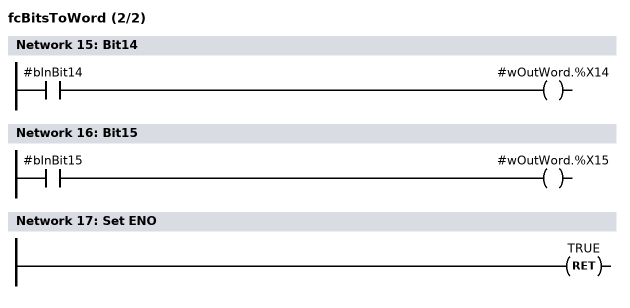
   RUNG wire#powerrail
      Contact( #bInBit14 )
      Coil( #wOutWord.%X14 )
   END_RUNG
   // the same network as SCL:
   #wOutWord.%X14 := #bInBit14;
END_REGION

REGION Network 16: Bit15
   RUNG wire#powerrail
      Contact( #bInBit15 )
      Coil( #wOutWord.%X15 )
   END_RUNG
   // the same network as SCL:
   #wOutWord.%X15 := #bInBit15;
END_REGION

REGION Network 17: Set ENO
   RUNG wire#powerrail
      ReturnCoil( TRUE )
   END_RUNG
   // the same network as SCL:
   ENO := TRUE;
   RETURN;
END_REGION
END_FUNCTION

FUNCTION_BLOCK "fbRoomFertigation"
{ S7_Optimized_Access := 'TRUE' }
VERSION : 0.1
   VAR_INPUT 
      arrInMutexRequests { ExternalAccessible := 'False'; ExternalVisible := 'False'; ExternalWritable := 'False'} : Array[0.."MAX_RACKS_PER_ROOM"] of Int;   // Array of mutex requests from racks
      arrInFertigationSettings { ExternalAccessible := 'False'; ExternalVisible := 'False'; ExternalWritable := 'False'} : Array[0.."MAX_RACKS_PER_ROOM"] of "udtFertigationSettings";
      rInTankLevel { ExternalAccessible := 'False'; ExternalVisible := 'False'; ExternalWritable := 'False'} : Real;
      rInNutrientALevel { ExternalAccessible := 'False'; ExternalVisible := 'False'; ExternalWritable := 'False'} : Real;
      rInNutrientBLevel { ExternalAccessible := 'False'; ExternalVisible := 'False'; ExternalWritable := 'False'} : Real;
      rInNutrientAcidLevel { ExternalAccessible := 'False'; ExternalVisible := 'False'; ExternalWritable := 'False'} : Real;
      rInpHSensor { ExternalAccessible := 'False'; ExternalVisible := 'False'; ExternalWritable := 'False'} : Real;
      rInECSensor { ExternalAccessible := 'False'; ExternalVisible := 'False'; ExternalWritable := 'False'} : Real;
      rInISESensor { ExternalAccessible := 'False'; ExternalVisible := 'False'; ExternalWritable := 'False'} : Real;
      rInORPReading { ExternalAccessible := 'False'; ExternalVisible := 'False'; ExternalWritable := 'False'} : Real;
      iInNumRacks { ExternalAccessible := 'False'; ExternalVisible := 'False'; ExternalWritable := 'False'} : Int;   // Number of racks to process mutex requests for
   END_VAR

   VAR_OUTPUT 
      bOutTankReturnSolenoid { ExternalAccessible := 'False'; ExternalVisible := 'False'; ExternalWritable := 'False'} : Bool;
      bOutMPathSolenoid { ExternalAccessible := 'False'; ExternalVisible := 'False'; ExternalWritable := 'False'} : Bool;
      bOutFreshWaterSolenoid { ExternalAccessible := 'False'; ExternalVisible := 'False'; ExternalWritable := 'False'} : Bool;
      bOutDischargeSolenoid { ExternalAccessible := 'False'; ExternalVisible := 'False'; ExternalWritable := 'False'} : Bool;
      bOutNutrientMixing { ExternalAccessible := 'False'; ExternalVisible := 'False'; ExternalWritable := 'False'} : Bool;
      bOutNutrientA { ExternalAccessible := 'False'; ExternalVisible := 'False'; ExternalWritable := 'False'} : Bool;
      bOutNutrientB { ExternalAccessible := 'False'; ExternalVisible := 'False'; ExternalWritable := 'False'} : Bool;
      bOutNutrientAcid { ExternalAccessible := 'False'; ExternalVisible := 'False'; ExternalWritable := 'False'} : Bool;
   END_VAR
   VAR_OUTPUT RETAIN
      arrOutNutrientReading { ExternalAccessible := 'False'; ExternalVisible := 'False'; ExternalWritable := 'False'} : Array[0.."MAX_RACKS_PER_ROOM"] of "udtNutrientReading";   // Array of nutrient readings going to racks
      arrOutMutexLocks { ExternalAccessible := 'False'; ExternalVisible := 'False'; ExternalWritable := 'False'} : Array[0.."MAX_RACKS_PER_ROOM"] of Int;   // Array of mutex locks going to racks
   END_VAR
   VAR_OUTPUT 
      arrOutSupplySolenoids { ExternalAccessible := 'False'; ExternalVisible := 'False'; ExternalWritable := 'False'} : Array[0.."MAX_RACKS_PER_ROOM"] of Bool;   // Array of supply solenoids for each rack
      arrOutReturnSolenoids { ExternalAccessible := 'False'; ExternalVisible := 'False'; ExternalWritable := 'False'} : Array[0.."MAX_RACKS_PER_ROOM"] of Bool;   // Array of return solenoids for each rack
   END_VAR

   VAR RETAIN
      Controls { ExternalVisible := 'False'} : Struct
         bPauseFertigation { ExternalVisible := 'False'} : Bool;   // While true, prevents next rack from locking
         rFloorPumpSpeedSP { ExternalVisible := 'False'} : Real;   // Floor pump speed (RPM)
         iNutrientMixingMode { ExternalVisible := 'False'} : Int;   // Nutrient mixing mode (0: off, 1: on, 2: 10 minute, 3: Continuous)
         rFreshLevelForMeasurementLoop { ExternalVisible := 'False'} : Real;   // Amount of fresh water to fill in the tank during rotate to clean measurement loop
         rFillLevelToPreviousShelf { ExternalVisible := 'False'} : Real := 8.0;   // Amount of water to push back to previous tank during return
         rReturnPathVolume { ExternalVisible := 'False'} : Real := 19.0;   // Return path volume (L) to fill from active rack
         rTankEmptyLevel { ExternalVisible := 'False'} : Real := 150.0;   // Volume at which tank is considered empty (L)
         rTankMaxVolume { ExternalVisible := 'False'} : Real := 900.0;   // Maximum volume for tank (L)
         bNutrientAgitation { ExternalVisible := 'False'} : Bool;
         tNutrientAgitationInterval { ExternalVisible := 'False'} : Time := T#60M;   // Agitation Frequency
         tNutrientAgitationDuration { ExternalVisible := 'False'} : Time := T#10M;   // Agitation Pump on-time
         rNutrientTanksLowerLimit { ExternalVisible := 'False'} : Real := 20.0;   // Liters
      END_STRUCT;
      Status { ExternalVisible := 'False'; ExternalWritable := 'False'} : Struct
         iState { ExternalVisible := 'False'; ExternalWritable := 'False'} : Int;   // Current operation (0: off, 1: Fill, 2:Measurement/Dosing, 3:Discharge)
         iActiveRack { ExternalVisible := 'False'; ExternalWritable := 'False'} : Int;   // Rack that currently has a lock, 0 if idle
         iLastMDRack { ExternalVisible := 'False'; ExternalWritable := 'False'} : Int;   // Keep track of previous rack for rotate and flush, 0 if previous operation was not measurement and dosing
      END_STRUCT;
      bTankReturnSolenoidCommand { ExternalAccessible := 'False'; ExternalVisible := 'False'; ExternalWritable := 'False'} : Bool;   // Command for tank return solenoid
      bMPathSolenoidCommand { ExternalAccessible := 'False'; ExternalVisible := 'False'; ExternalWritable := 'False'} : Bool;   // Command for measurement path solenoid
      bFreshWaterSolenoidCommand { ExternalAccessible := 'False'; ExternalVisible := 'False'; ExternalWritable := 'False'} : Bool;   // Command for fresh water solenoid
      bDischargeSolenoidCommand { ExternalAccessible := 'False'; ExternalVisible := 'False'; ExternalWritable := 'False'} : Bool;   // Command for discharge solenoid
      bNutrientMixingCommand { ExternalAccessible := 'False'; ExternalVisible := 'False'; ExternalWritable := 'False'} : Bool;   // Command for nutrient mixing enable
      bNutrientACommand { ExternalAccessible := 'False'; ExternalVisible := 'False'; ExternalWritable := 'False'} : Bool;   // Command for dosing nutrient A
      bNutrientBCommand { ExternalAccessible := 'False'; ExternalVisible := 'False'; ExternalWritable := 'False'} : Bool;   // Command for dosing nutrient B
      bNutrientAcidCommand { ExternalAccessible := 'False'; ExternalVisible := 'False'; ExternalWritable := 'False'} : Bool;
      TON_Discharge {InstructionName := 'TON_TIME'; LibVersion := '1.0'; S7_SetPoint := 'False'} : TON_TIME;
      TON_24HourNutrientMix {InstructionName := 'TON_TIME'; LibVersion := '1.0'; ExternalAccessible := 'False'; ExternalVisible := 'False'; ExternalWritable := 'False'; S7_SetPoint := 'False'} : TON_TIME;
   END_VAR
   VAR 
      fbRoomMeasurementDosing { ExternalAccessible := 'False'; ExternalVisible := 'False'; ExternalWritable := 'False'; S7_SetPoint := 'False'} : "fbRoomMeasurementDosing";
   END_VAR
   VAR RETAIN
      bTransferring { ExternalAccessible := 'False'; ExternalVisible := 'False'; ExternalWritable := 'False'} : Bool;   // Memory bit for transfer to rack during fill process
      rTransferredVolume { ExternalAccessible := 'False'; ExternalVisible := 'False'; ExternalWritable := 'False'} : Real;
      rVolumeToTransfer { ExternalAccessible := 'False'; ExternalVisible := 'False'; ExternalWritable := 'False'} : Real;
      bEndDischarge { ExternalAccessible := 'False'; ExternalVisible := 'False'; ExternalWritable := 'False'} : Bool;
   END_VAR
   VAR 
      TON_PeriodicNutrientAgitation {InstructionName := 'TON_TIME'; LibVersion := '1.0'} : TON_TIME;
      TP_PeriodicNutrientAgitation {InstructionName := 'TP_TIME'; LibVersion := '1.0'} : TP_TIME;
   END_VAR

   VAR_TEMP 
      bFoundActive : Bool;
      i : Int;   // Iterable for mutex request 
      tCurrentDateTime : Date_And_Time;   // Current PLC Date and Time
      tCurrentTime : Time_Of_Day;   // Current PLC Time of Day
      retVal : Int;   // Garbage return value from RD_LOC_T
      bMDDone : Bool;
      rTargetFillVolume : Real;
   END_VAR

   VAR CONSTANT 
      eRoomMode_Off : Int := 0;   // Room Off State
      eRoomMode_Fill : Int := 1;   // Room Filling State
      eRoomMode_MeasurementDosing : Int := 2;   // Room Measurement and Dosing State
      eRoomMode_Discharge : Int := 3;   // Room Discharge State
      eNutrientMixingMode_Off : Int := 0;   // Forced off
      eNutrientMixingMode_On : Int := 1;   // Forced on
      eNutrientMixingMode_Periodic : Int := 2;   // Run according to Interval/Duration settings
      eNutrientMixingMode_FullDay : Int := 3;   // Run for 24 hours then switch to Ten Minute mode
      MIX_START_TIME : Time_Of_Day := TOD#12:00:00;   // Start of 10 minute mix at noon
      MIX_END_TIME : Time_Of_Day := TOD#12:10:00;   // End of 10 minute mix at noon
   END_VAR


BEGIN
	REGION 0: Off
	    // Close all solenoids
	    // Iterate through mutex requests to trigger state change
	    // Send lock when mutex request arrives
	    
	    IF #Status.iState = #eRoomMode_Off THEN
	        #bTankReturnSolenoidCommand := 0;
	        #bMPathSolenoidCommand := 0;
	        #bFreshWaterSolenoidCommand := 0;
	        
	        #bFoundActive := 0;
	        IF NOT #Controls.bPauseFertigation THEN // if not paused, check for next rack requesting lock
	            FOR #i := 1 TO #iInNumRacks DO
	                IF #arrInMutexRequests[#i] <> #eRoomMode_Off THEN
	                    
	                    // Mutex request active - update state and active rack, send lock
	                    #Status.iState := #arrInMutexRequests[#i];
	                    #Status.iActiveRack := #i;
	                    #arrOutMutexLocks[#i] := #Status.iState;
	                    #bFoundActive := 1;
	                    //Break out of for loop
	                    EXIT;
	                END_IF;
	            END_FOR;
	        END_IF;
	        IF NOT #bFoundActive THEN
	            #Status.iActiveRack := 0;
	        END_IF;
	    END_IF;
	    
	    
	END_REGION
	
	REGION 1: Fill
	    // Open fresh water solenoid, fill until max volume reached or rack volume reached, close fresh water solenoid
	    // Open rack supply solenoid, activate floor pump, wait for main tank content to return to rack
	    
	    // Need to keep track of how much has been sent to the rack, until total volume added matches OperatingVolume + TotalShelfVolume or
	    // resevoir reaches max volume
	    
	    IF #Status.iState = #eRoomMode_Fill THEN
	        
	        #Status.iLastMDRack := 0; // no rotate if last rack last rack was filled
	        
	        #rTargetFillVolume := #arrInFertigationSettings[#Status.iActiveRack].rOperatingVolume
	        + #arrInFertigationSettings[#Status.iActiveRack].rTotalShelfVolume;
	        
	        IF #rTransferredVolume >= #rTargetFillVolume OR
	            #arrInFertigationSettings[#Status.iActiveRack].rRackCurrentVolume > #arrInFertigationSettings[#Status.iActiveRack].rMaxReservoirVolume THEN
	            // Full volume or rack reservoir is too full, done with fill
	            #Status.iState := #eRoomMode_Off;
	            #arrOutMutexLocks[#Status.iActiveRack] := 0;
	            
	            #arrOutSupplySolenoids[#Status.iActiveRack] := 0;
	            #bFreshWaterSolenoidCommand := 0;
	            
	            #bTransferring := 0;
	            #rTransferredVolume := 0;
	            
	            
	        ELSIF #rInTankLevel < #Controls.rTankMaxVolume AND
	            #rInTankLevel - #Controls.rTankEmptyLevel + #rTransferredVolume < #rTargetFillVolume AND
	            NOT #bTransferring THEN
	            // Adding water to the main tank
	            #bFreshWaterSolenoidCommand := 1;
	            
	        ELSIF NOT #bTransferring THEN
	            // Start transfer from main tank to rack
	            #bTransferring := 1;
	            #bFreshWaterSolenoidCommand := 0;
	            #rVolumeToTransfer := #rInTankLevel - #Controls.rTankEmptyLevel;
	            
	        END_IF;
	        
	        IF #bTransferring AND #rInTankLevel <= #Controls.rTankEmptyLevel THEN
	            // Transfer is done, add volume to transferred total
	            #bTransferring := 0;
	            #rTransferredVolume += #rVolumeToTransfer;
	            #rVolumeToTransfer := 0;
	            #arrOutSupplySolenoids[#Status.iActiveRack] := 0;
	            
	        END_IF;
	        
	        // Transfer from main tank to rack until main tank is empty
	        #arrOutSupplySolenoids[#Status.iActiveRack] := #bTransferring;
	        
	    END_IF;
	    
	    
	END_REGION
	
	
	REGION 2: Measurement AND Dosing
	    // Call measurement and dosing subfunction for the room
	    // Only write to outputs when in the correct mode
	    
	    // Reset the last rack id to skip rotate if that rack is not accepting rotate
	    IF #Status.iState = #eRoomMode_MeasurementDosing AND #Status.iLastMDRack <> 0 THEN
	        IF NOT #arrInFertigationSettings[#Status.iLastMDRack].bEnableIncomingRotate THEN
	            #Status.iLastMDRack := 0;
	        END_IF;
	    END_IF;
	    
	     #fbRoomMeasurementDosing(bInStart := (#Status.iState = #eRoomMode_MeasurementDosing),
	                              iInActiveRack := #Status.iActiveRack,
	                              iInPreviousRack := #Status.iLastMDRack,
	                              rInTankLevel := #rInTankLevel,
	                              rInRackLevel := #arrInFertigationSettings[#Status.iActiveRack].rRackCurrentVolume,
	                              rInISEReading := #rInISESensor,
	                              rInECReading := #rInECSensor,
	                              rInpHReading := #rInpHSensor,
	                              rInORPReading := #rInORPReading,
	                              rInFillLevelToPreviousShelf := #Controls.rFillLevelToPreviousShelf,
	                              rInFreshLevelForMLoop := #Controls.rFreshLevelForMeasurementLoop,
	                              rInReturnPathVolume := #Controls.rReturnPathVolume,
	                              rInTankEmptyLevel := #Controls.rTankEmptyLevel,
	                              InFertigationSettings := #arrInFertigationSettings[#Status.iActiveRack],
	                              bOutTankReturnSolenoidCommand => #fbRoomMeasurementDosing.bOutTankReturnSolenoidCommand,
	                              bOutActiveRackReturnSolenoidCommand => #fbRoomMeasurementDosing.bOutActiveRackReturnSolenoidCommand,
	                              bOutActiveRackSupplySolenoidCommand => #fbRoomMeasurementDosing.bOutActiveRackSupplySolenoidCommand,
	                              bOutPreviousRackReturnSolenoidCommand => #fbRoomMeasurementDosing.bOutPreviousRackReturnSolenoidCommand,
	                              bOutPreviousRackSupplySolenoidCommand => #fbRoomMeasurementDosing.bOutPreviousRackSupplySolenoidCommand,
	                              bOutFreshWaterSolenoidCommand => #fbRoomMeasurementDosing.bOutFreshWaterSolenoidCommand,
	                              bOutDischargeSolenoidCommand => #fbRoomMeasurementDosing.bOutDischargeSolenoidCommand,
	                              bOutMPathSolenoidCommand => #fbRoomMeasurementDosing.bOutMPathSolenoidCommand,
	                              bOutNutrientACommand => #fbRoomMeasurementDosing.bOutNutrientACommand,
	                              bOutNutrientBCommand => #fbRoomMeasurementDosing.bOutNutrientBCommand,
	                              OutNutrientReadings => #fbRoomMeasurementDosing.OutNutrientReadings,
	                              bOutDone => #bMDDone);
	    
	    //Handle output writing
	    IF #Status.iState = #eRoomMode_MeasurementDosing THEN
	        #bTankReturnSolenoidCommand := #fbRoomMeasurementDosing.bOutTankReturnSolenoidCommand;
	        #bFreshWaterSolenoidCommand := #fbRoomMeasurementDosing.bOutFreshWaterSolenoidCommand;
	        #bDischargeSolenoidCommand := #fbRoomMeasurementDosing.bOutDischargeSolenoidCommand;
	        #bMPathSolenoidCommand := #fbRoomMeasurementDosing.bOutMPathSolenoidCommand;
	        #bNutrientACommand := #fbRoomMeasurementDosing.bOutNutrientACommand;
	        #bNutrientBCommand := #fbRoomMeasurementDosing.bOutNutrientBCommand;
	        #arrOutReturnSolenoids[#Status.iActiveRack] := #fbRoomMeasurementDosing.bOutActiveRackReturnSolenoidCommand;
	        #arrOutSupplySolenoids[#Status.iActiveRack] := #fbRoomMeasurementDosing.bOutActiveRackSupplySolenoidCommand;
	        #arrOutReturnSolenoids[#Status.iLastMDRack] := #fbRoomMeasurementDosing.bOutPreviousRackReturnSolenoidCommand;
	        #arrOutSupplySolenoids[#Status.iLastMDRack] := #fbRoomMeasurementDosing.bOutPreviousRackSupplySolenoidCommand;
	        #arrOutNutrientReading[#Status.iActiveRack] := #fbRoomMeasurementDosing.OutNutrientReadings;
	        
	        IF #bMDDone THEN
	            #Status.iState := #eRoomMode_Off;
	            #arrOutMutexLocks[#Status.iActiveRack] := #eRoomMode_Off;
	            #Status.iLastMDRack := #Status.iActiveRack; // save rack id for rotate on next M&D
	        END_IF;
	    END_IF;
	    
	END_REGION
	
	REGION 3: Discharge
	    // Open discharge solenoid and rack's return solenoid
	    // Wait for discharge time
	    // Close solenoids and release lock
	    // Return to Off mode
	    
	    #TON_Discharge(IN := (#Status.iState = #eRoomMode_Discharge),
	                   PT := #arrInFertigationSettings[#Status.iActiveRack].tDischargeTime);
	    
	    IF #Status.iState = #eRoomMode_Discharge THEN
	        
	        IF #TON_Discharge.Q OR #arrInFertigationSettings[#Status.iActiveRack].bEndDischargeCommand THEN
	            #bEndDischarge := 1;
	        END_IF;
	        
	        
	        IF #bEndDischarge THEN
	            #arrOutMutexLocks[#Status.iActiveRack] := #eRoomMode_Off;
	            
	            // wait until pump stops to close valves
	            IF #arrInFertigationSettings[#Status.iActiveRack].bPumpAtStandstill THEN 
	                #bDischargeSolenoidCommand := 0;
	                #arrOutReturnSolenoids[#Status.iActiveRack] := 0;
	                #Status.iLastMDRack := 0; // no rotate if last rack was discharged
	                #Status.iState := #eRoomMode_Off;
	                #bEndDischarge := 0;
	                #TON_Discharge.IN := 0; // reset timer
	            END_IF;
	            
	        ELSE
	            #bDischargeSolenoidCommand := 1;
	            #arrOutReturnSolenoids[#Status.iActiveRack] := 1;
	            
	        END_IF;
	        
	    END_IF;
	    
	END_REGION
	
	REGION Nutrient Tank Mixing
	    // 0: forced off, 1: forced on, 2: 10 minutes per day at noon, 3: Run for 24 hours then jump to mode 2
	    
	    
	    // if the tanks are too low, switch agitation to off
	    (*IF #rInNutrientALevel < #Controls.rNutrientTanksLowerLimit OR #rInNutrientBLevel < #Controls.rNutrientTanksLowerLimit THEN
	        #Controls.iNutrientMixingMode := #eNutrientMixingMode_Off;
	    END_IF;
	    *)
	    
	    #TON_24HourNutrientMix(IN := (#Controls.iNutrientMixingMode = #eNutrientMixingMode_FullDay),
	                           PT := T#24h);
	    
	    // if mode is set to periodic agitation, run timer to periodically run pumps
	    #Controls.bNutrientAgitation := #TON_PeriodicNutrientAgitation.Q;
	    #TON_PeriodicNutrientAgitation(IN := #Controls.iNutrientMixingMode = #eNutrientMixingMode_Periodic AND NOT #Controls.bNutrientAgitation,
	                                   PT := #Controls.tNutrientAgitationInterval);
	    
	    #TP_PeriodicNutrientAgitation(IN := #Controls.bNutrientAgitation,
	                                  PT := #Controls.tNutrientAgitationDuration,
	                                  Q => #bNutrientMixingCommand);
	    
	    
	    IF #Controls.iNutrientMixingMode = #eNutrientMixingMode_Off THEN
	        #bNutrientMixingCommand := 0;
	        
	    ELSIF #Controls.iNutrientMixingMode = #eNutrientMixingMode_On THEN
	        #bNutrientMixingCommand := 1;
	        
	        (*
	    ELSIF #Controls.iNutrientMixingMode = #eNutrientMixingMode_Periodic THEN
	      
	        // Extract current PLC time
	        #retVal := RD_LOC_T(OUT => #tCurrentDateTime);
	        #tCurrentTime := DT_TO_TOD(IN := #tCurrentDateTime);
	        
	        IF (#tCurrentTime < #MIX_END_TIME) AND (#tCurrentTime > #MIX_START_TIME) T
	            #bNutrientMixingCommand := 1;
	        ELSE
	            #bNutrientMixingCommand := 0;
	        END_IF;
	        
	        *)
	        
	    ELSIF #Controls.iNutrientMixingMode = #eNutrientMixingMode_FullDay THEN
	        
	        IF #TON_24HourNutrientMix.Q THEN
	            #bNutrientMixingCommand := 0;
	            #Controls.iNutrientMixingMode := #eNutrientMixingMode_Periodic;
	        ELSE
	            #bNutrientMixingCommand := 1;
	        END_IF;
	        
	        // Catchall for incorrectly entered state, just turn off mixer
	    //ELSE
	    //    #bNutrientMixingCommand := 0;
	    END_IF;
	    
	    // IF not forced on and then tank levels are too low, override above and disable mixing until tanks are filled
	    IF NOT (#Controls.iNutrientMixingMode = #eNutrientMixingMode_On) AND
	           (#rInNutrientALevel < #Controls.rNutrientTanksLowerLimit OR
	            #rInNutrientBLevel < #Controls.rNutrientTanksLowerLimit) THEN
	        #bNutrientMixingCommand := 0;
	    END_IF;
	    
	END_REGION
	
	REGION Set digital outputs
	    #bOutTankReturnSolenoid := #bTankReturnSolenoidCommand;
	    #bOutMPathSolenoid      := #bMPathSolenoidCommand;
	    #bOutFreshWaterSolenoid := #bFreshWaterSolenoidCommand;
	    #bOutDischargeSolenoid  := #bDischargeSolenoidCommand;
	    #bOutNutrientMixing     := #bNutrientMixingCommand;
	    #bOutNutrientA          := #bNutrientACommand;
	    #bOutNutrientB          := #bNutrientBCommand;
	    #bOutNutrientAcid       := #bNutrientAcidCommand;
	    
	END_REGION
	
	
	
END_FUNCTION_BLOCK

FUNCTION_BLOCK "fbRoomMeasurementDosing"
{ S7_Optimized_Access := 'TRUE' }
VERSION : 0.1
   VAR_INPUT 
      bInStart { ExternalAccessible := 'False'; ExternalVisible := 'False'; ExternalWritable := 'False'} : Bool;   // Start command for sequence
      iInActiveRack { ExternalAccessible := 'False'; ExternalVisible := 'False'; ExternalWritable := 'False'} : Int;   // Current rack requesting MD
      iInPreviousRack { ExternalAccessible := 'False'; ExternalVisible := 'False'; ExternalWritable := 'False'} : Int;   // Previous rack, if last operation was also MD (0 otherwise)
      rInTankLevel { ExternalAccessible := 'False'; ExternalVisible := 'False'; ExternalWritable := 'False'} : Real;   // Current tank level (L)
      rInISEReading { ExternalAccessible := 'False'; ExternalVisible := 'False'; ExternalWritable := 'False'} : Real;   // Current ISE sensor level
      rInECReading { ExternalAccessible := 'False'; ExternalVisible := 'False'; ExternalWritable := 'False'} : Real;   // Current EC sensor level
      rInpHReading { ExternalAccessible := 'False'; ExternalVisible := 'False'; ExternalWritable := 'False'} : Real;   // Current pH sensor level
      rInORPReading { ExternalAccessible := 'False'; ExternalVisible := 'False'; ExternalWritable := 'False'} : Real;
      rInRackLevel { ExternalAccessible := 'False'; ExternalVisible := 'False'; ExternalWritable := 'False'} : Real;   // Current rack reservoir level
      rInFreshLevelForMLoop { ExternalAccessible := 'False'; ExternalVisible := 'False'; ExternalWritable := 'False'} : Real;
      rInFillLevelToPreviousShelf { ExternalAccessible := 'False'; ExternalVisible := 'False'; ExternalWritable := 'False'} : Real;
      rInReturnPathVolume { ExternalAccessible := 'False'; ExternalVisible := 'False'; ExternalWritable := 'False'} : Real;   // Return path volume (L) to fill from active rack
      rInTankEmptyLevel { ExternalAccessible := 'False'; ExternalVisible := 'False'; ExternalWritable := 'False'} : Real;   // Volume at which tank is considered empty (L)
      InFertigationSettings { ExternalAccessible := 'False'; ExternalVisible := 'False'; ExternalWritable := 'False'} : "udtFertigationSettings";   // Current rack fertigation settings
   END_VAR

   VAR_OUTPUT RETAIN
      bOutTankReturnSolenoidCommand { ExternalAccessible := 'False'; ExternalVisible := 'False'; ExternalWritable := 'False'} : Bool;   // Output for writing to tank return solenoid
      bOutActiveRackReturnSolenoidCommand { ExternalAccessible := 'False'; ExternalVisible := 'False'; ExternalWritable := 'False'} : Bool;
      bOutActiveRackSupplySolenoidCommand { ExternalAccessible := 'False'; ExternalVisible := 'False'; ExternalWritable := 'False'} : Bool;
      bOutPreviousRackReturnSolenoidCommand { ExternalAccessible := 'False'; ExternalVisible := 'False'; ExternalWritable := 'False'} : Bool;
      bOutPreviousRackSupplySolenoidCommand { ExternalAccessible := 'False'; ExternalVisible := 'False'; ExternalWritable := 'False'} : Bool;
      bOutFreshWaterSolenoidCommand { ExternalAccessible := 'False'; ExternalVisible := 'False'; ExternalWritable := 'False'} : Bool;
      bOutDischargeSolenoidCommand { ExternalAccessible := 'False'; ExternalVisible := 'False'; ExternalWritable := 'False'} : Bool;
      bOutMPathSolenoidCommand { ExternalAccessible := 'False'; ExternalVisible := 'False'; ExternalWritable := 'False'} : Bool;
      bOutNutrientACommand { ExternalAccessible := 'False'; ExternalVisible := 'False'; ExternalWritable := 'False'} : Bool;   // Output for writing to Nutrient A enable
      bOutNutrientBCommand { ExternalAccessible := 'False'; ExternalVisible := 'False'; ExternalWritable := 'False'} : Bool;   // Output for writing to Nutrient B enable
      OutNutrientReadings { ExternalAccessible := 'False'; ExternalVisible := 'False'; ExternalWritable := 'False'} : "udtNutrientReading";   // Final measured sensor levels for rack
      bOutDone { ExternalAccessible := 'False'; ExternalVisible := 'False'; ExternalWritable := 'False'} : Bool;
   END_VAR

   VAR RETAIN
      iState { ExternalAccessible := 'False'; ExternalVisible := 'False'; ExternalWritable := 'False'} : Int;
      iNextState { ExternalAccessible := 'False'; ExternalVisible := 'False'; ExternalWritable := 'False'} : Int;
      rTankStartingLevel { ExternalAccessible := 'False'; ExternalVisible := 'False'; ExternalWritable := 'False'} : Real;
      TON_MeasurementTimer {InstructionName := 'TON_TIME'; LibVersion := '1.0'; ExternalAccessible := 'False'; ExternalVisible := 'False'; ExternalWritable := 'False'; S7_SetPoint := 'False'} : TON_TIME;
      TON_NutrientATimer {InstructionName := 'TON_TIME'; LibVersion := '1.0'; ExternalAccessible := 'False'; ExternalVisible := 'False'; ExternalWritable := 'False'; S7_SetPoint := 'False'} : TON_TIME;
      TON_NutrientBTimer {InstructionName := 'TON_TIME'; LibVersion := '1.0'; ExternalAccessible := 'False'; ExternalVisible := 'False'; ExternalWritable := 'False'; S7_SetPoint := 'False'} : TON_TIME;
   END_VAR
   VAR 
      TON_TankLowLimitTimer {InstructionName := 'TON_TIME'; LibVersion := '1.0'} : TON_TIME;
   END_VAR

   VAR CONSTANT 
      eMDState_Idle : Int;
      eMDState_Rotate_Start : Int := 100;
      eMDState_Rotate_FillTankFromRack : Int := 102;
      eMDState_Rotate_PushToPrevious : Int := 104;
      eMDState_Rotate_FillTankFresh : Int := 106;
      eMDState_Rotate_MeasurementLoop : Int := 108;
      eMDState_Rotate_Done : Int := 119;
      eMDState_Measure_Start : Int := 120;
      eMDState_Measure_FillTankFromRack : Int := 122;
      eMDState_Measure_OpenMLoop : Int := 124;
      eMDState_Measure_Done : Int := 139;
      eMDState_Dosing_Start : Int := 140;
      eMDState_Dosing_AddNutrientA : Int := 142;
      eMDState_Dosing_AddNutrientB : Int := 144;
      eMDState_Dosing_AddFreshWater : Int := 146;
      eMDState_Dosing_Done : Int := 159;
      eMDState_Return_Start : Int := 160;
      eMDState_Return_FillPreviousRack : Int := 162;
      eMDState_Return_FillActiveRack : Int := 164;
      eMDState_Return_CloseSupplyPath : Int := 166;
      eMDState_Return_Done : Int := 169;
      iISEMode_Off : Int := 0;
      iISEMode_Load : Int := 1;
      iISEMode_Deplete : Int := 2;
   END_VAR


BEGIN
	REGION State 0: Idle
	    // Wait for start command to move on to rotate if a previous rack used the piping 
	    //  or directly to measure if not 
	    
	    IF #iState = #eMDState_Idle THEN
	        #bOutDone := 0;
	        IF #bInStart THEN
	            IF #iInPreviousRack = 0 OR #iInPreviousRack = #iInActiveRack THEN
	                #iNextState := #eMDState_Measure_Start;
	            ELSE
	                #iNextState := #eMDState_Rotate_Start;
	            END_IF;
	        END_IF;
	    END_IF;
	        
	    
	END_REGION
	
	REGION State 100: Rotate
	    // Open the tank return solenoid
	    // Open the return solenoid and close the shelf solenoid for the current rack until a fixed amount of water is pumped into the tank
	    // Close the return solenoid of the current rack and open the supply valve of the previous rack to push 19L from the 
	    //     tank into the previous rack. 
	    //     
	    
	    // Open tank return and rack return, close shelf, record starting tank level, then move to next state
	    IF #iState = #eMDState_Rotate_Start THEN
	        #bOutTankReturnSolenoidCommand := 1; 
	        #bOutActiveRackReturnSolenoidCommand := 1;
	        #iNextState := #eMDState_Rotate_FillTankFromRack;
	        #rTankStartingLevel := #rInTankLevel;
	    END_IF;
	    
	    // Once the target fill level is reached, close the return solenoids, open the previous rack's supply, then move to next state
	    IF #iState = #eMDState_Rotate_FillTankFromRack THEN
	        IF #rInTankLevel >= #rTankStartingLevel + #rInReturnPathVolume  OR #rInRackLevel <= #InFertigationSettings.rMinReservoirVolume THEN
	            #bOutActiveRackReturnSolenoidCommand := 0;
	            #bOutPreviousRackSupplySolenoidCommand := 1;
	            #bOutTankReturnSolenoidCommand := 1;
	            #iNextState := #eMDState_Rotate_PushToPrevious;
	        END_IF;
	    END_IF;
	    
	    // Run until 19L have been pushed into the previous rack and the tank is back at its original level, then close the
	    // previous rack's supply solenoid and move to next state
	    IF #iState = #eMDState_Rotate_PushToPrevious THEN
	        
	        IF #rInTankLevel <= #rTankStartingLevel * 1.2 THEN // HACK
	            #bOutPreviousRackSupplySolenoidCommand := 0;
	            #iNextState := #eMDState_Rotate_FillTankFresh;
	        END_IF;
	        
	    END_IF;
	    
	    // Open the fresh water supply and fill the tank until the target level is reached, then close the fresh water supply, open the
	    // measurement path solenoid and the discharge solenoid and move to the next state
	    IF #iState = #eMDState_Rotate_FillTankFresh THEN
	        
	        IF #rInTankLevel >= #rTankStartingLevel + #rInFreshLevelForMLoop THEN
	            #bOutFreshWaterSolenoidCommand := 0;
	            #bOutMPathSolenoidCommand := 1;
	            #bOutDischargeSolenoidCommand := 1;
	            #bOutTankReturnSolenoidCommand := 0;
	            #iNextState := #eMDState_Rotate_MeasurementLoop;
	        ELSE
	            #bOutFreshWaterSolenoidCommand := 1;
	        END_IF;
	    END_IF;
	    
	    // Push water out through the measurement loop. Once the tank is empty, close measurement path solenoid and
	    // the discharge solenoid and move to the next state
	    IF #iState = #eMDState_Rotate_MeasurementLoop THEN
	        
	        IF #rInTankLevel <= #rInTankEmptyLevel THEN
	            
	            #bOutMPathSolenoidCommand := 0;
	            #bOutDischargeSolenoidCommand := 0;
	            #iNextState := #eMDState_Rotate_Done;
	        END_IF;
	    END_IF;
	    
	    IF #iState = #eMDState_Rotate_Done THEN
	        #iNextState := #eMDState_Measure_Start;
	    END_IF;
	    
	END_REGION
	
	REGION State 120: Measure
	    // Receive water from rack and start measurement phase. Open measurement loop, push water through, record sensor readings, 
	    // determine setpoints, and move on to dosing
	    
	    #TON_MeasurementTimer(IN := (#iState = #eMDState_Measure_OpenMLoop),
	                         PT := #InFertigationSettings.tMeasurementTime);
	    
	    // Open tank return and shelf return solenoid
	    IF #iState = #eMDState_Measure_Start THEN
	        #bOutTankReturnSolenoidCommand := 1;
	        #bOutActiveRackReturnSolenoidCommand := 1;
	        #iNextState := #eMDState_Measure_FillTankFromRack;
	        #rTankStartingLevel := #rInTankLevel;
	    END_IF;
	    
	    // Wait to receive target level from rack, close rack return solenoid
	    IF #iState = #eMDState_Measure_FillTankFromRack THEN
	        IF #rInTankLevel >= (#InFertigationSettings.rMeasurementVolume + #rInTankEmptyLevel) OR
	            #rInRackLevel <= #InFertigationSettings.rMinReservoirVolume THEN
	            #iNextState := #eMDState_Measure_OpenMLoop;
	            #bOutActiveRackReturnSolenoidCommand := 0;
	        END_IF;
	    END_IF;
	    
	    // Open MPath solenoid, wait for measurement time then record measurement
	    IF #iState = #eMDState_Measure_OpenMLoop THEN
	        
	        IF #TON_MeasurementTimer.Q THEN
	            #OutNutrientReadings.rISEReading := #rInISEReading;
	            #OutNutrientReadings.rECReading := #rInECReading;
	            #OutNutrientReadings.rpHReading := #rInpHReading;
	            #OutNutrientReadings.rORPReading := #rInORPReading;
	            #bOutMPathSolenoidCommand := 0;
	            #bOutTankReturnSolenoidCommand := 0;
	            #iNextState := #eMDState_Measure_Done;
	        ELSE
	            #bOutMPathSolenoidCommand := 1;
	        END_IF;
	    END_IF;
	    
	    
	    IF #iState = #eMDState_Measure_Done THEN
	        #iNextState := #eMDState_Dosing_Start;
	    END_IF;
	   
	    
	END_REGION
	
	REGION State 140: Dosing
	    
	    // Check if rack fertigation logic has requested dosing
	    // Add enabled nutrients one at a time for dosing time then add fresh water to tank
	    
	    IF #iState = #eMDState_Dosing_Start THEN
	        
	        IF #InFertigationSettings.bDosingActive THEN
	            
	            IF #InFertigationSettings.bNutrientAEnable THEN
	                #iNextState := #eMDState_Dosing_AddNutrientA;
	            ELSIF #InFertigationSettings.bNutrientBEnable THEN
	                #iNextState := #eMDState_Dosing_AddNutrientB;
	            ELSE
	                #iNextState := #eMDState_Dosing_AddFreshWater;
	            END_IF;
	            
	        ELSE
	            #iNextState := #eMDState_Dosing_AddFreshWater;
	        END_IF;
	    END_IF;
	    
	    #TON_NutrientATimer(IN := (#iState = #eMDState_Dosing_AddNutrientA),
	                       PT := #InFertigationSettings.tNutrientDosingDuration);
	    // Add nutrient A for dosing time, then check if nutrient B is needed
	    IF #iState = #eMDState_Dosing_AddNutrientA THEN
	        
	        IF #TON_NutrientATimer.Q THEN
	            #bOutNutrientACommand := 0;
	            IF #InFertigationSettings.bNutrientBEnable THEN
	                #iNextState := #eMDState_Dosing_AddNutrientB;
	            ELSE
	                #iNextState := #eMDState_Dosing_AddFreshWater;
	            END_IF;
	        ELSE
	            #bOutNutrientACommand := 1;
	        END_IF;
	    END_IF;
	    
	    #TON_NutrientBTimer(IN := (#iState = #eMDState_Dosing_AddNutrientB),
	                       PT := #InFertigationSettings.tNutrientDosingDuration);
	    // Add nutrient B for dosing time, then move on to water fill
	    IF #iState = #eMDState_Dosing_AddNutrientB THEN
	        
	        IF #TON_NutrientBTimer.Q THEN
	            #bOutNutrientBCommand := 0;
	            #iNextState := #eMDState_Dosing_AddFreshWater;
	        ELSE
	            #bOutNutrientBCommand := 1;
	        END_IF;
	    END_IF;
	    
	    // Add fresh water to tank if tank level plus rack is less than the operating volume
	    IF #iState = #eMDState_Dosing_AddFreshWater THEN
	        IF (#rInTankLevel - #rInTankEmptyLevel + #rInRackLevel < #InFertigationSettings.rOperatingVolume) THEN
	            #bOutFreshWaterSolenoidCommand := 1;
	        ELSE
	            #bOutFreshWaterSolenoidCommand := 0;
	            #iNextState := #eMDState_Dosing_Done;
	        END_IF;
	    END_IF;
	    
	    
	    IF #iState = #eMDState_Dosing_Done THEN
	        #iNextState := #eMDState_Return_Start;
	    END_IF;
	    
	END_REGION
	
	REGION State 160: Return TO Tank
	    // If a previous rack was used, open supply path to previous rack, wait for 8L drop in tank
	    // Open supply path to active rack, activate floor pump, wait for tank contents to return to rack
	    // Close supply path
	    
	    // Determine which rack to start return to
	    IF #iState = #eMDState_Return_Start THEN
	        
	        IF #iInPreviousRack = 0 OR #iInPreviousRack = #iInActiveRack  THEN
	            #iNextState := #eMDState_Return_FillActiveRack;
	        ELSE
	            #iNextState := #eMDState_Return_FillPreviousRack;
	        END_IF;
	        #rTankStartingLevel := #rInTankLevel;
	    END_IF;
	    
	    // Open supply path to previous rack, wait for 8L drop in tank, close previous rack return path
	    IF #iState = #eMDState_Return_FillPreviousRack THEN
	        #bOutPreviousRackSupplySolenoidCommand := 1;
	        IF #rInTankLevel < (#rTankStartingLevel - #rInFillLevelToPreviousShelf) THEN
	            #bOutPreviousRackSupplySolenoidCommand := 0;
	            #iNextState := #eMDState_Return_FillActiveRack;
	        END_IF;
	    END_IF;
	    
	    // Open supply path to active rack
	    IF #iState = #eMDState_Return_FillActiveRack THEN
	        #rTankStartingLevel := #rInTankLevel;
	        #bOutActiveRackSupplySolenoidCommand := 1;
	        #iNextState := #eMDState_Return_CloseSupplyPath;
	    END_IF;
	    
	    // Wait for tank to empty, close supply path
	    //#TON_TankLowLimitTimer(IN:=#rInTankLevel <= #rInTankEmptyLevel,
	    //                       PT:=T#3s);
	    IF #iState = #eMDState_Return_CloseSupplyPath THEN
	        IF #rInTankLevel <= #rInTankEmptyLevel * 1.2 OR #rInRackLevel >= #InFertigationSettings.rMaxReservoirVolume THEN // HACK
	            #bOutActiveRackSupplySolenoidCommand := 0;
	            #iNextState := #eMDState_Return_Done;
	        END_IF;
	    END_IF;
	    
	    //Return to Idle at end of M&D
	    IF #iState = #eMDState_Return_Done THEN
	        #bOutDone := 1;
	        #iNextState := #eMDState_Idle;
	    END_IF;
	    
	END_REGION
	
	
	REGION Update State
	    IF #iState <> #iNextState THEN
	        #iState := #iNextState;
	    END_IF;
	END_REGION
	
	
END_FUNCTION_BLOCK

FUNCTION_BLOCK "fbRoomHVAC"   // FB2, LAD
{ S7_Optimized_Access := 'TRUE' }
VERSION : 0.1
// stored: AutoNumber true, IsIECCheckEnabled false, IsRetainMemResEnabled false, MemoryReserve 100, SetENOAutomatically false, UDAEnableTagReadback false
   VAR_INPUT
      iInCO2ReadingRaw { ExternalAccessible := 'False'; ExternalVisible := 'False'; ExternalWritable := 'False'} : Int;
   END_VAR
   VAR_OUTPUT
      bOutCO2Solenoid { ExternalAccessible := 'False'; ExternalVisible := 'False'; ExternalWritable := 'False'} : Bool;
   END_VAR
   VAR
      Temperature_Cooling { ExternalVisible := 'False'} : "fbAlarmedSetpoint";
      Humidity { ExternalVisible := 'False'} : "fbAlarmedSetpoint";
   END_VAR
   VAR RETAIN
      Controls { ExternalVisible := 'False'} : Struct
         rHeatingSP { ExternalVisible := 'False'} : Real := 55.0;
         bResetAlarm { ExternalVisible := 'False'} : Bool;
         bResetModbus { ExternalVisible := 'False'} : Bool;
         rDehum_SAT_SP { ExternalVisible := 'False'} : Real := 65.0;
         rDehum_MOD_SP { ExternalVisible := 'False'} : Real := 60.0;
      END_STRUCT;
      Status { ExternalVisible := 'False'; ExternalWritable := 'False'} : Struct
         SupplyAirTemperature { ExternalVisible := 'False'; ExternalWritable := 'False'} : Real;
         bModbusError { ExternalVisible := 'False'; ExternalWritable := 'False'} : Bool;
         wLastModbusErrorCode { ExternalVisible := 'False'; ExternalWritable := 'False'} : Word;
         Compressor_1_Percentage { ExternalVisible := 'False'; ExternalWritable := 'False'} : Real;
         Compressor_2_Percentage { ExternalVisible := 'False'; ExternalWritable := 'False'} : Real;
         ZoneAirEnthalpy { ExternalVisible := 'False'; ExternalWritable := 'False'} : Real;
         Compressor_1_Command { ExternalVisible := 'False'; ExternalWritable := 'False'} : Bool;
         Compressor_1_Enabled { ExternalVisible := 'False'; ExternalWritable := 'False'} : Bool;
         Compressor_1_Alarm { ExternalVisible := 'False'; ExternalWritable := 'False'} : Bool;
         Compressor_2_Command { ExternalVisible := 'False'; ExternalWritable := 'False'} : Bool;
         Compressor_2_Enabled { ExternalVisible := 'False'; ExternalWritable := 'False'} : Bool;
         Compressor_2_Alarm { ExternalVisible := 'False'; ExternalWritable := 'False'} : Bool;
         LPS1_Alarm { ExternalVisible := 'False'; ExternalWritable := 'False'} : Bool;
         LPS2_Alarm { ExternalVisible := 'False'; ExternalWritable := 'False'} : Bool;
         HPS1_Alarm { ExternalVisible := 'False'; ExternalWritable := 'False'} : Bool;
         HPS2_Alarm { ExternalVisible := 'False'; ExternalWritable := 'False'} : Bool;
         Dehum_1_Enabled { ExternalVisible := 'False'; ExternalWritable := 'False'} : Bool;
         Dehum_2_Enabled { ExternalVisible := 'False'; ExternalWritable := 'False'} : Bool;
         HGRH_Modulation { ExternalVisible := 'False'; ExternalWritable := 'False'} : Real;
         Freeze_Alarm_1 { ExternalVisible := 'False'; ExternalWritable := 'False'} : Bool;
         Freeze_Alarm_2 { ExternalVisible := 'False'; ExternalWritable := 'False'} : Bool;
         DX_LAT_1 { ExternalVisible := 'False'; ExternalWritable := 'False'} : Real;
         DX_LAT_2 { ExternalVisible := 'False'; ExternalWritable := 'False'} : Real;
      END_STRUCT;
      Config { ExternalVisible := 'False'} : Struct
         ModbusServerAddr { ExternalVisible := 'False'} : IP_V4;   // IP address for Modbus TCP server
         ID { ExternalVisible := 'False'} : UInt := 81;   // Unique ID for connection, also used as port number on PLC
      END_STRUCT;
   END_VAR
   VAR
      CO2Control { ExternalVisible := 'False'} : "fbRoomCO2Control";
      TCPConnection { ExternalAccessible := 'False'; ExternalVisible := 'False'; ExternalWritable := 'False'} : TCON_IP_v4;
      fbModbusTCPClient_Instance { ExternalAccessible := 'False'; ExternalVisible := 'False'; ExternalWritable := 'False'} : "fbModbusTCPClient";
      Read_Discrete { ExternalAccessible := 'False'; ExternalVisible := 'False'; ExternalWritable := 'False'} : Array[0..13] of "udtModbusValBool";
      Write_Discrete { ExternalAccessible := 'False'; ExternalVisible := 'False'; ExternalWritable := 'False'} : Array[0..0] of "udtModbusValBool";
      Read_Registers { ExternalAccessible := 'False'; ExternalVisible := 'False'; ExternalWritable := 'False'} : Array[0..9] of "udtModbusValReal";
      Write_Registers { ExternalAccessible := 'False'; ExternalVisible := 'False'; ExternalWritable := 'False'} : Array[0..4] of "udtModbusValReal";
      TON_ModbusReset { S7_SetPoint := 'True'} : TON_TIME;
      mbreset { ExternalAccessible := 'False'; ExternalVisible := 'False'; ExternalWritable := 'False'} : Bool;
      TP_ModbusResetPulse { S7_SetPoint := 'True'} : TP_TIME;
   END_VAR
   VAR CONSTANT
      cFakeScaling : Int := 150;
      cRoomTempIndex : Int := 0;
      cHumidityIndex : Int := 1;
      cCO2Index : Int := 2;
      cSupplyAirTempIndex : Int := 3;
   END_VAR
   // Temperature_Cooling.arrSetpoints[1].rSetpoint := 75.0;
   // Humidity.arrSetpoints[1].rSetpoint := 55.0;
   // Config.ModbusServerAddr.ADDR[1] := 10;
   // Config.ModbusServerAddr.ADDR[2] := 1;
   // Config.ModbusServerAddr.ADDR[3] := 0;
   // Config.ModbusServerAddr.ADDR[4] := 20;
   // TCPConnection.ConnectionType := 11;
   // TCPConnection.ActiveEstablished := true;
   // TCPConnection.RemoteAddress.ADDR[1] := 10;
   // TCPConnection.RemoteAddress.ADDR[2] := 1;
   // TCPConnection.RemoteAddress.ADDR[3] := 0;
   // TCPConnection.RemoteAddress.ADDR[4] := 20;
   // TCPConnection.RemotePort := 502;
   // TCPConnection.LocalPort := 1001;
BEGIN

REGION Network 1 (SCL): Set connection parameters
   #TCPConnection.InterfaceId := "Local~PROFINET_interface_1"; // PLC ethernet port
   #TCPConnection.ID := UINT_TO_WORD(#Config.ID);
   #TCPConnection.ConnectionType := 11; // TCP
   #TCPConnection.ActiveEstablished := TRUE;
   #TCPConnection.RemoteAddress := #Config.ModbusServerAddr;
   #TCPConnection.RemotePort := 502; // Default for Modbus TCP
   #TCPConnection.LocalPort := #Config.ID;
END_REGION

REGION Network 2 (SCL): Reset Modbus on Error

   #mbreset := #TON_ModbusReset.Q;
   #TON_ModbusReset(IN := #Status.bModbusError AND NOT #mbreset,
                    PT := T#10S);

   #TP_ModbusResetPulse(IN:=#mbreset,
                        PT:=T#5S,
                        Q => #Controls.bResetModbus);

   (*

   IF #Status.bModbusError AND NOT #mbreset THEN
       #Controls.bResetModbus := 1;
       //#mbreset := 1;
   END_IF;

   IF #TON_ModbusReset.Q AND #Controls.bResetModbus THEN
       #Controls.bResetModbus := 0;
       #TON_ModbusReset.IN := 0;
       //#mbreset := 0;
   END_IF;
   *)
END_REGION

REGION Network 3 (SCL): Set up registers
   // Read coils and discrete inputs (00001 and 10001)
   #Read_Discrete[0].iAddr := 10048; // Compressor_1_Command
   #Read_Discrete[1].iAddr := 10067; // Compressor_1_Enabled
   #Read_Discrete[2].iAddr := 10091; // Compressor_1_Alarm
   #Read_Discrete[3].iAddr := 10049; // Compressor_2_Command
   #Read_Discrete[4].iAddr := 10008; // Compressor_2_Enabled
   #Read_Discrete[5].iAddr := 10068; // Compressor_2_Alarm
   #Read_Discrete[6].iAddr := 10089; // LPS1_Alarm
   #Read_Discrete[7].iAddr := 10034; // LPS2_Alarm
   #Read_Discrete[8].iAddr := 10093; // HPS1_Alarm
   #Read_Discrete[9].iAddr := 10097; // HPS2_Alarm
   #Read_Discrete[10].iAddr := 10019; // Dehum_1_Enabled
   #Read_Discrete[11].iAddr := 10014; // Dehum_2_Enabled
   #Read_Discrete[12].iAddr := 10090; // Freeze Alarm #1
   #Read_Discrete[13].iAddr := 10037; // Freeze Alarm #2

   // Write coils (00001)
   #Write_Discrete[0].iAddr := 00020; // Alarm reset
   #Write_Discrete[0].bVal := #Controls.bResetAlarm;

   // Read input and holding registers (30001 and 40001)
   #Read_Registers[cRoomTempIndex].iRegister      := 30035; // Room Temperature
   #Read_Registers[cHumidityIndex].iRegister      := 30031; // Humidity
   #Read_Registers[cCO2Index].iRegister := 30031;//30001; // CO2
   #Read_Registers[cSupplyAirTempIndex].iRegister := 30043; // Supply Air Temperature

   #Read_Registers[4].iRegister := 30077; // Compressor_1_percentage
   #Read_Registers[5].iRegister := 30077;//30049; // Compressor_2_percentage
   #Read_Registers[6].iRegister := 30039; // ZoneAirEnthalpy
   #Read_Registers[7].iRegister := 30095; //HGRH_Modulation
   #Read_Registers[8].iRegister := 30013; // DX_LAT #1
   #Read_Registers[9].iRegister := 30087; // DX_LAT #2

   // Write holding registers (40001)
   #Write_Registers[0].iRegister := 40119; // Cooling SP
   #Write_Registers[0].rVal := #Temperature_Cooling.rSetpoint;

   #Write_Registers[1].iRegister := 40121; // Heating SP
   #Write_Registers[1].rVal := #Controls.rHeatingSP;

   #Write_Registers[2].iRegister := 40039; // Dehumidification SP
   #Write_Registers[2].rVal := #Humidity.rSetpoint;

   #Write_Registers[3].iRegister := 40043; // Dehum Supply Air SP
   #Write_Registers[3].rVal := #Controls.rDehum_SAT_SP;

   #Write_Registers[4].iRegister := 40097; // Dehumidification MOD SP... DX LAT SP? degrees F?
   #Write_Registers[4].rVal := #Controls.rDehum_MOD_SP;
   (*
   #Write_Data[3].iRegister := 2; // CO2 SP 1
   #Write_Data[3].rVal := #CO2.rSetpoint;

   #Write_Data[4].iRegister := 66; // CO2 SP 2
   #Write_Data[4].rVal := #CO2.rSetpoint;
   *)
END_REGION

REGION Network 4: Modbus TCP Client Block Call
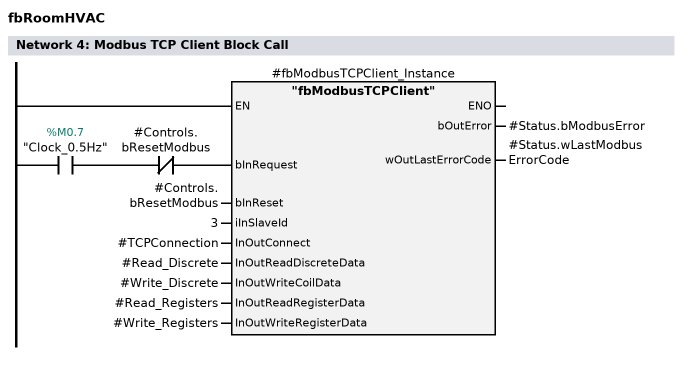
   RUNG wire#powerrail
      #fbModbusTCPClient_Instance(bInRequest := wire#w1, bInReset := #Controls.bResetModbus, iInSlaveId := 3, InOutConnect := #TCPConnection, InOutReadDiscreteData := #Read_Discrete, InOutWriteCoilData := #Write_Discrete, InOutReadRegisterData := #Read_Registers, InOutWriteRegisterData := #Write_Registers, bOutError => #Status.bModbusError, wOutLastErrorCode => #Status.wLastModbusErrorCode)
   END_RUNG
   RUNG wire#powerrail
      Contact( "Clock_0.5Hz" )
      I_Contact( #Controls.bResetModbus )
   END_RUNG wire#w1
   // the same network as SCL:
   #fbModbusTCPClient_Instance(bInRequest := "Clock_0.5Hz" AND NOT #Controls.bResetModbus,   // "fbModbusTCPClient"
                           bInReset := #Controls.bResetModbus,
                           iInSlaveId := 3,
                           InOutConnect := #TCPConnection,
                           InOutReadDiscreteData := #Read_Discrete,
                           InOutWriteCoilData := #Write_Discrete,
                           InOutReadRegisterData := #Read_Registers,
                           InOutWriteRegisterData := #Write_Registers,
                           bOutError => #Status.bModbusError,
                           wOutLastErrorCode => #Status.wLastModbusErrorCode);
END_REGION

REGION Network 5 (SCL): Parse received data
   // Status data
   #Status.Compressor_1_Percentage := #Read_Registers[4].rVal;
   #Status.Compressor_2_Percentage := #Read_Registers[5].rVal;
   #Status.ZoneAirEnthalpy := #Read_Registers[6].rVal;
   #Status.HGRH_Modulation := #Read_Registers[7].rVal;
   #Status.DX_LAT_1 := #Read_Registers[8].rVal;
   #Status.DX_LAT_2 := #Read_Registers[9].rVal;


   #Status.Compressor_1_Command := #Read_Discrete[0].bVal;
   #Status.Compressor_1_Enabled := #Read_Discrete[1].bVal;
   #Status.Compressor_1_Alarm :=   #Read_Discrete[2].bVal;
   #Status.Compressor_2_Command := #Read_Discrete[3].bVal;
   #Status.Compressor_2_Enabled := #Read_Discrete[4].bVal;
   #Status.Compressor_2_Alarm :=   #Read_Discrete[5].bVal;
   #Status.LPS1_Alarm := #Read_Discrete[6].bVal;
   #Status.LPS2_Alarm := #Read_Discrete[7].bVal;
   #Status.HPS1_Alarm := #Read_Discrete[8].bVal;
   #Status.HPS2_Alarm := #Read_Discrete[9].bVal;
   #Status.Dehum_1_Enabled := #Read_Discrete[10].bVal;
   #Status.Dehum_2_Enabled := #Read_Discrete[11].bVal;
   #Status.Freeze_Alarm_1 := #Read_Discrete[12].bVal;
   #Status.Freeze_Alarm_2 := #Read_Discrete[13].bVal;


   // Bypass analog scaling for alarmed setpoints
   #Temperature_Cooling.Config.rLowCalibration := 0;
   #Temperature_Cooling.Config.rHighCalibration := #cFakeScaling;
   #Humidity.Config.rLowCalibration := 0;
   #Humidity.Config.rHighCalibration := #cFakeScaling;

   #Temperature_Cooling(
                        iInRawValue := REAL_TO_INT(#Read_Registers[cRoomTempIndex].rVal /
                                                   #cFakeScaling * "IoScaling.S7Analog.Default.iRawMax"));

   #Humidity(
             iInRawValue := REAL_TO_INT(#Read_Registers[cHumidityIndex].rVal /
                                        #cFakeScaling * "IoScaling.S7Analog.Default.iRawMax"));

   #Status.SupplyAirTemperature := #Read_Registers[cSupplyAirTempIndex].rVal;
END_REGION

REGION Network 6 (SCL): Call CO2 control logic
   #CO2Control(iInCO2ReadingRaw := #iInCO2ReadingRaw,
               bOutSolenoid=>#bOutCO2Solenoid);
END_REGION
END_FUNCTION_BLOCK

FUNCTION_BLOCK "fbModbusTCPClient"   // FB12, LAD
{ S7_Optimized_Access := 'TRUE' }
VERSION : 0.1
// stored: AutoNumber true, IsIECCheckEnabled false, IsRetainMemResEnabled false, MemoryReserve 100, SetENOAutomatically false, UDAEnableTagReadback false
   VAR_INPUT
      bInRequest { ExternalAccessible := 'False'; ExternalVisible := 'False'; ExternalWritable := 'False'} : Bool;
      bInReset { ExternalVisible := 'False'} : Bool;
      iInSlaveId { ExternalAccessible := 'False'; ExternalVisible := 'False'; ExternalWritable := 'False'} : UInt;
   END_VAR
   VAR_OUTPUT
      bOutError { ExternalAccessible := 'False'; ExternalVisible := 'False'; ExternalWritable := 'False'} : Bool;
      wOutLastErrorCode { ExternalAccessible := 'False'; ExternalVisible := 'False'; ExternalWritable := 'False'} : Word;
   END_VAR
   VAR_IN_OUT
      InOutConnect : TCON_IP_v4;
      InOutReadDiscreteData : Array[*] of "udtModbusValBool";
      InOutWriteCoilData : Array[*] of "udtModbusValBool";
      InOutReadRegisterData : Array[*] of "udtModbusValReal";
      InOutWriteRegisterData : Array[*] of "udtModbusValReal";
   END_VAR
   VAR
      iState { ExternalAccessible := 'False'; ExternalVisible := 'False'; ExternalWritable := 'False'} : Int;
      iNextState { ExternalAccessible := 'False'; ExternalVisible := 'False'; ExternalWritable := 'False'} : Int;
      insModbusClient_TCP { ExternalAccessible := 'False'; ExternalVisible := 'False'; ExternalWritable := 'False'} : MB_CLIENT;
      bTrigReset { ExternalAccessible := 'False'; ExternalVisible := 'False'; ExternalWritable := 'False'} : Bool;
      bTrigReq { ExternalAccessible := 'False'; ExternalVisible := 'False'; ExternalWritable := 'False'} : Bool;
      iNumReadRegisters { ExternalAccessible := 'False'; ExternalVisible := 'False'; ExternalWritable := 'False'} : DInt;
      iNumWriteRegisters { ExternalAccessible := 'False'; ExternalVisible := 'False'; ExternalWritable := 'False'} : DInt;
      iCurrentRegisterReadIndex { ExternalAccessible := 'False'; ExternalVisible := 'False'; ExternalWritable := 'False'} : DInt;
      iCurrentRegisterWriteIndex { ExternalAccessible := 'False'; ExternalVisible := 'False'; ExternalWritable := 'False'} : DInt;
      arrDataWords { ExternalAccessible := 'False'; ExternalVisible := 'False'; ExternalWritable := 'False'} : Array[0..1] of Word;
      iNumReadDiscrete { ExternalAccessible := 'False'; ExternalVisible := 'False'; ExternalWritable := 'False'} : DInt;
      iCurrentDiscreteReadIndex { ExternalAccessible := 'False'; ExternalVisible := 'False'; ExternalWritable := 'False'} : DInt;
      iCurrentCoilWriteIndex { ExternalAccessible := 'False'; ExternalVisible := 'False'; ExternalWritable := 'False'} : DInt;
      iNumWriteCoils { ExternalAccessible := 'False'; ExternalVisible := 'False'; ExternalWritable := 'False'} : DInt;
   END_VAR
   VAR_TEMP
      iMode : USInt;
      iDataAddr : UDInt;
      tempDWord : DWord;
      bConnect : Bool;
      rTemp : Real;
   END_VAR
   VAR CONSTANT
      MODE_READ : USInt := 0;
      MODE_WRITE : USInt := 1;
      IDLE : Int := 0;
      READ_DISC_INIT : Int := 100;
      READ_DISC : Int := 110;
      READ_DISC_NEXT : Int := 120;
      WRITE_COILS_INIT : Int := 200;
      WRITE_COILS : Int := 210;
      WRITE_COILS_NEXT : Int := 220;
      READ_REGS_INIT : Int := 300;
      READ_REGS : Int := 310;
      READ_REGS_PARSE : Int := 320;
      READ_REGS_NEXT : Int := 330;
      WRITE_REGS_INIT : Int := 400;
      WRITE_REGS : Int := 410;
      WRITE_REGS_READBACK_INIT : Int := 420;
      WRITE_REGS_READBACK : Int := 430;
      WRITE_REGS_READBACK_PARSE : Int := 440;
      WRITE_REGS_NEXT : Int := 450;
   END_VAR
   VAR_TEMP   // added for the SCL form of the ladder/FBD networks
      _w1 : Bool;
      _w2 : Bool;
      _w3 : Bool;
      _w4 : Bool;
      _w5 : Bool;
      _w6 : Bool;
      _w7 : Bool;
      _w8 : Bool;
   END_VAR
BEGIN

REGION Network 1: ------------------------------ State Logic ----------------------------------
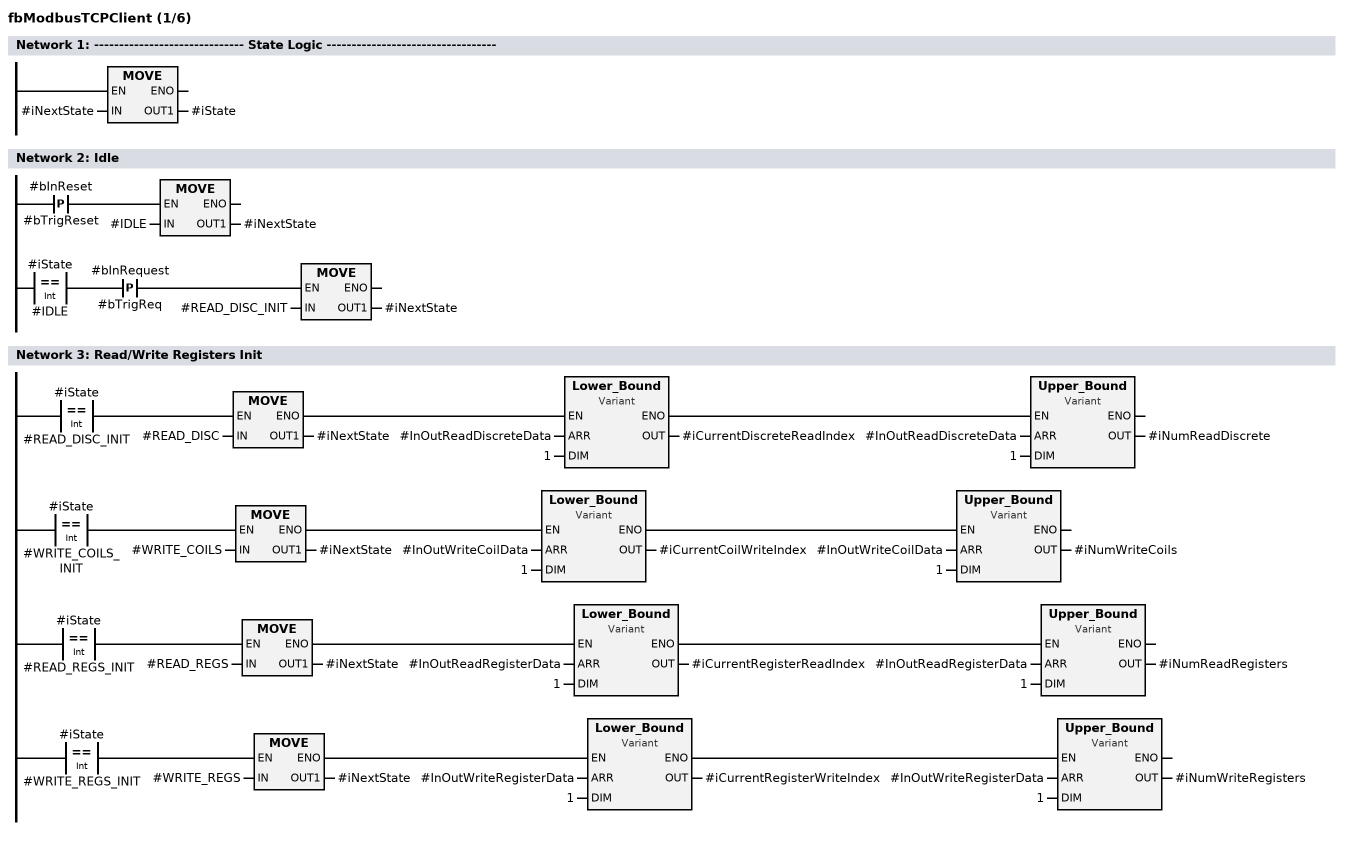
   RUNG wire#powerrail
      Move(in := #iNextState, out1 => #iState)
   END_RUNG
   // the same network as SCL:
   #iState := #iNextState;
END_REGION

REGION Network 2: Idle
   RUNG wire#powerrail
      P_Contact(operand := #bInReset, bit := #bTrigReset)
      Move(in := #IDLE, out1 => #iNextState)
   END_RUNG
   RUNG wire#powerrail
      { S7_Templates := "SrcType := Int" } EQ_Contact(in1 := #iState, in2 := #IDLE)
      P_Contact(operand := #bInRequest, bit := #bTrigReq)
      Move(in := #READ_DISC_INIT, out1 => #iNextState)
   END_RUNG
   // the same network as SCL:
   #_w1 := #bInReset AND NOT #bTrigReset;   // rising edge of #bInReset
   #bTrigReset := #bInReset;
   IF #_w1 THEN #iNextState := #IDLE; END_IF;
   #_w2 := (#iState = #IDLE) AND #bInRequest AND NOT #bTrigReq;   // rising edge of #bInRequest
   #bTrigReq := #bInRequest;
   IF #_w2 THEN #iNextState := #READ_DISC_INIT; END_IF;
END_REGION

REGION Network 3: Read/Write Registers Init
   // no SCL statement known for Lower_Bound, Upper_Bound: written as a call
   // ENO of a box is taken as its EN; it also drops when the box reports an error
   IF #iState = #READ_DISC_INIT THEN
       #iNextState := #READ_DISC;
       Lower_Bound(arr := #InOutReadDiscreteData, dim := 1, out => #iCurrentDiscreteReadIndex);
       Upper_Bound(arr := #InOutReadDiscreteData, dim := 1, out => #iNumReadDiscrete);
   END_IF;
   IF #iState = #WRITE_COILS_INIT THEN
       #iNextState := #WRITE_COILS;
       Lower_Bound(arr := #InOutWriteCoilData, dim := 1, out => #iCurrentCoilWriteIndex);
       Upper_Bound(arr := #InOutWriteCoilData, dim := 1, out => #iNumWriteCoils);
   END_IF;
   IF #iState = #READ_REGS_INIT THEN
       #iNextState := #READ_REGS;
       Lower_Bound(arr := #InOutReadRegisterData, dim := 1, out => #iCurrentRegisterReadIndex);
       Upper_Bound(arr := #InOutReadRegisterData, dim := 1, out => #iNumReadRegisters);
   END_IF;
   IF #iState = #WRITE_REGS_INIT THEN
       #iNextState := #WRITE_REGS;
       Lower_Bound(arr := #InOutWriteRegisterData, dim := 1, out => #iCurrentRegisterWriteIndex);
       Upper_Bound(arr := #InOutWriteRegisterData, dim := 1, out => #iNumWriteRegisters);
   END_IF;
END_REGION

REGION Network 4: Wait for Read/Write to be done
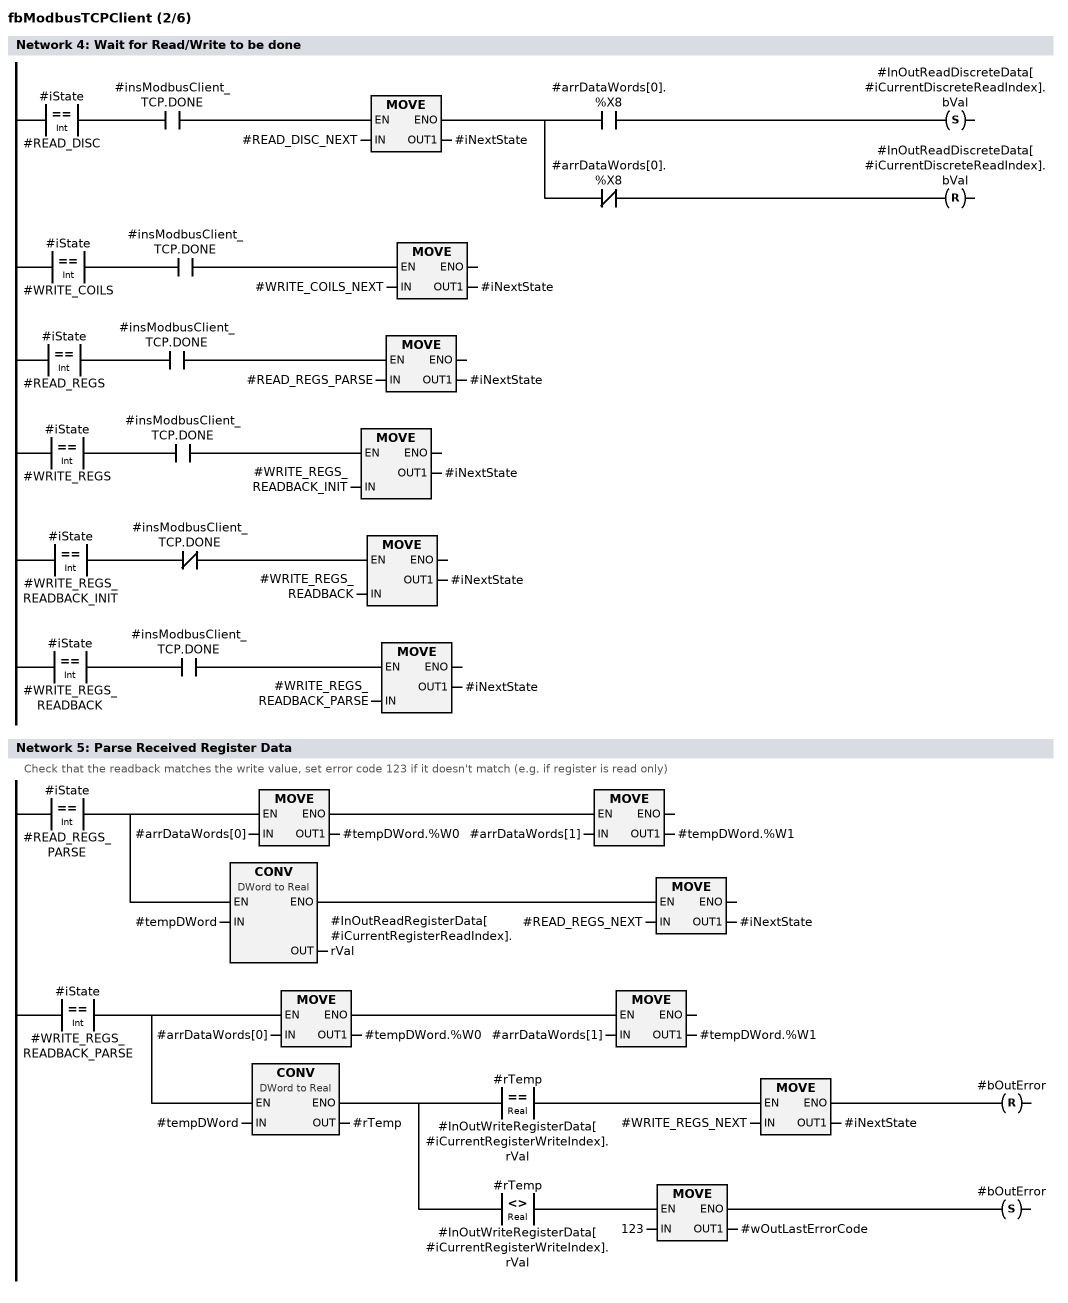
   RUNG wire#powerrail
      { S7_Templates := "SrcType := Int" } EQ_Contact(in1 := #iState, in2 := #READ_DISC)
      Contact( #insModbusClient_TCP.DONE )
      Move(in := #READ_DISC_NEXT, out1 => #iNextState)
      wire#w1
      Contact( #arrDataWords[0].%X8 )
      S_Coil( #InOutReadDiscreteData[#iCurrentDiscreteReadIndex].bVal )
   END_RUNG
   RUNG wire#w1
      I_Contact( #arrDataWords[0].%X8 )
      R_Coil( #InOutReadDiscreteData[#iCurrentDiscreteReadIndex].bVal )
   END_RUNG
   RUNG wire#powerrail
      { S7_Templates := "SrcType := Int" } EQ_Contact(in1 := #iState, in2 := #WRITE_COILS)
      Contact( #insModbusClient_TCP.DONE )
      Move(in := #WRITE_COILS_NEXT, out1 => #iNextState)
   END_RUNG
   RUNG wire#powerrail
      { S7_Templates := "SrcType := Int" } EQ_Contact(in1 := #iState, in2 := #READ_REGS)
      Contact( #insModbusClient_TCP.DONE )
      Move(in := #READ_REGS_PARSE, out1 => #iNextState)
   END_RUNG
   RUNG wire#powerrail
      { S7_Templates := "SrcType := Int" } EQ_Contact(in1 := #iState, in2 := #WRITE_REGS)
      Contact( #insModbusClient_TCP.DONE )
      Move(in := #WRITE_REGS_READBACK_INIT, out1 => #iNextState)
   END_RUNG
   RUNG wire#powerrail
      { S7_Templates := "SrcType := Int" } EQ_Contact(in1 := #iState, in2 := #WRITE_REGS_READBACK_INIT)
      I_Contact( #insModbusClient_TCP.DONE )
      Move(in := #WRITE_REGS_READBACK, out1 => #iNextState)
   END_RUNG
   RUNG wire#powerrail
      { S7_Templates := "SrcType := Int" } EQ_Contact(in1 := #iState, in2 := #WRITE_REGS_READBACK)
      Contact( #insModbusClient_TCP.DONE )
      Move(in := #WRITE_REGS_READBACK_PARSE, out1 => #iNextState)
   END_RUNG
   // the same network as SCL:
   #_w1 := (#iState = #READ_DISC) AND #insModbusClient_TCP.DONE;
   IF #_w1 THEN #iNextState := #READ_DISC_NEXT; END_IF;
   IF #_w1 AND #arrDataWords[0].%X8 THEN
       #InOutReadDiscreteData[#iCurrentDiscreteReadIndex].bVal := TRUE;
   END_IF;
   IF #_w1 AND NOT #arrDataWords[0].%X8 THEN
       #InOutReadDiscreteData[#iCurrentDiscreteReadIndex].bVal := FALSE;
   END_IF;
   IF (#iState = #WRITE_COILS) AND #insModbusClient_TCP.DONE THEN #iNextState := #WRITE_COILS_NEXT; END_IF;
   IF (#iState = #READ_REGS) AND #insModbusClient_TCP.DONE THEN #iNextState := #READ_REGS_PARSE; END_IF;
   IF (#iState = #WRITE_REGS) AND #insModbusClient_TCP.DONE THEN
       #iNextState := #WRITE_REGS_READBACK_INIT;
   END_IF;
   IF (#iState = #WRITE_REGS_READBACK_INIT) AND NOT #insModbusClient_TCP.DONE THEN
       #iNextState := #WRITE_REGS_READBACK;
   END_IF;
   IF (#iState = #WRITE_REGS_READBACK) AND #insModbusClient_TCP.DONE THEN
       #iNextState := #WRITE_REGS_READBACK_PARSE;
   END_IF;
END_REGION

REGION Network 5: Parse Received Register Data
   // Check that the readback matches the write value, set error code 123 if it doesn't match (e.g. if register is read only)
   RUNG wire#powerrail
      { S7_Templates := "SrcType := Int" } EQ_Contact(in1 := #iState, in2 := #READ_REGS_PARSE)
      wire#w1
      Move(in := #arrDataWords[0], out1 => #tempDWord.%W0)
      Move(in := #arrDataWords[1], out1 => #tempDWord.%W1)
   END_RUNG
   RUNG wire#w1
      { S7_Templates := "[SrcType := DWord, DestType := Real]" } Convert(in := #tempDWord, out => #InOutReadRegisterData[#iCurrentRegisterReadIndex].rVal)
      Move(in := #READ_REGS_NEXT, out1 => #iNextState)
   END_RUNG
   RUNG wire#powerrail
      { S7_Templates := "SrcType := Int" } EQ_Contact(in1 := #iState, in2 := #WRITE_REGS_READBACK_PARSE)
      wire#w2
      Move(in := #arrDataWords[0], out1 => #tempDWord.%W0)
      Move(in := #arrDataWords[1], out1 => #tempDWord.%W1)
   END_RUNG
   RUNG wire#w2
      { S7_Templates := "[SrcType := DWord, DestType := Real]" } Convert(in := #tempDWord, out => #rTemp)
      wire#w3
      { S7_Templates := "SrcType := Real" } EQ_Contact(in1 := #rTemp, in2 := #InOutWriteRegisterData[#iCurrentRegisterWriteIndex].rVal)
      Move(in := #WRITE_REGS_NEXT, out1 => #iNextState)
      R_Coil( #bOutError )
   END_RUNG
   RUNG wire#w3
      { S7_Templates := "SrcType := Real" } NE_Contact(in1 := #rTemp, in2 := #InOutWriteRegisterData[#iCurrentRegisterWriteIndex].rVal)
      Move(in := 123, out1 => #wOutLastErrorCode)
      S_Coil( #bOutError )
   END_RUNG
   // the same network as SCL:
   IF #iState = #READ_REGS_PARSE THEN
       #tempDWord.%W0 := #arrDataWords[0];
       #tempDWord.%W1 := #arrDataWords[1];
       #InOutReadRegisterData[#iCurrentRegisterReadIndex].rVal := DWORD_TO_REAL(#tempDWord);
       #iNextState := #READ_REGS_NEXT;
   END_IF;
   #_w1 := #iState = #WRITE_REGS_READBACK_PARSE;
   IF #_w1 THEN
       #tempDWord.%W0 := #arrDataWords[0];
       #tempDWord.%W1 := #arrDataWords[1];
       #rTemp := DWORD_TO_REAL(#tempDWord);
   END_IF;
   IF #_w1 AND (#rTemp = #InOutWriteRegisterData[#iCurrentRegisterWriteIndex].rVal) THEN
       #iNextState := #WRITE_REGS_NEXT;
       #bOutError := FALSE;
   END_IF;
   IF #_w1 AND (#rTemp <> #InOutWriteRegisterData[#iCurrentRegisterWriteIndex].rVal) THEN
       #wOutLastErrorCode := 123;
       #bOutError := TRUE;
   END_IF;
END_REGION

REGION Network 6: Move on to next address
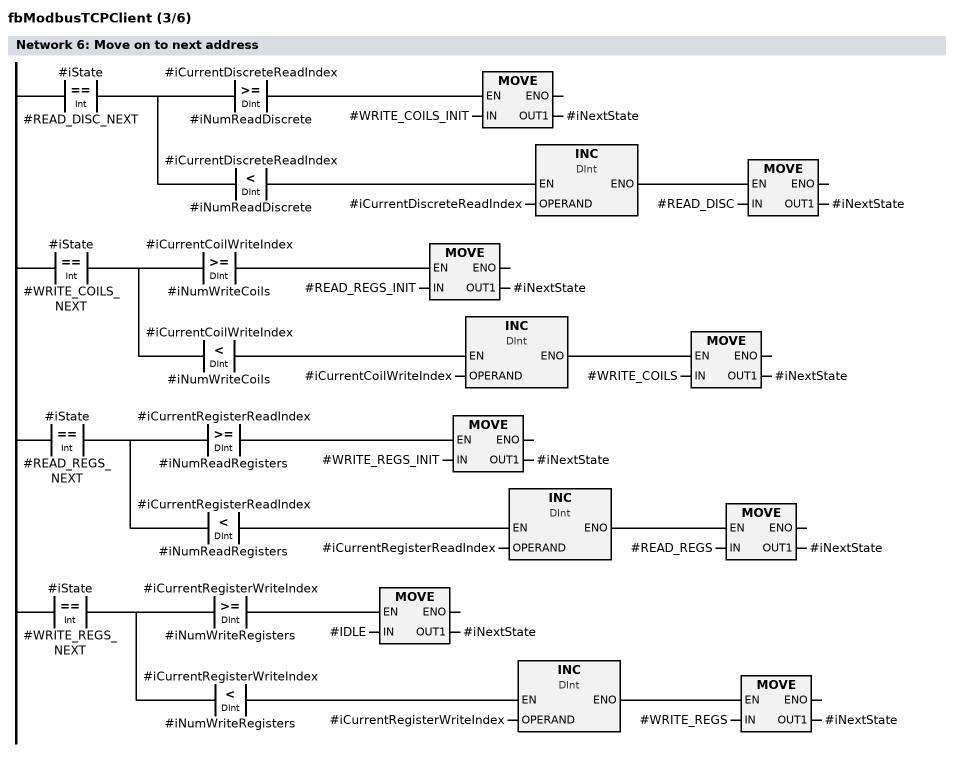
   RUNG wire#powerrail
      { S7_Templates := "SrcType := Int" } EQ_Contact(in1 := #iState, in2 := #READ_DISC_NEXT)
      wire#w1
      { S7_Templates := "SrcType := DInt" } GE_Contact(in1 := #iCurrentDiscreteReadIndex, in2 := #iNumReadDiscrete)
      Move(in := #WRITE_COILS_INIT, out1 => #iNextState)
   END_RUNG
   RUNG wire#w1
      { S7_Templates := "SrcType := DInt" } LT_Contact(in1 := #iCurrentDiscreteReadIndex, in2 := #iNumReadDiscrete)
      { S7_Templates := "DestType := DInt" } Inc( #iCurrentDiscreteReadIndex )
      Move(in := #READ_DISC, out1 => #iNextState)
   END_RUNG
   RUNG wire#powerrail
      { S7_Templates := "SrcType := Int" } EQ_Contact(in1 := #iState, in2 := #WRITE_COILS_NEXT)
      wire#w2
      { S7_Templates := "SrcType := DInt" } GE_Contact(in1 := #iCurrentCoilWriteIndex, in2 := #iNumWriteCoils)
      Move(in := #READ_REGS_INIT, out1 => #iNextState)
   END_RUNG
   RUNG wire#w2
      { S7_Templates := "SrcType := DInt" } LT_Contact(in1 := #iCurrentCoilWriteIndex, in2 := #iNumWriteCoils)
      { S7_Templates := "DestType := DInt" } Inc( #iCurrentCoilWriteIndex )
      Move(in := #WRITE_COILS, out1 => #iNextState)
   END_RUNG
   RUNG wire#powerrail
      { S7_Templates := "SrcType := Int" } EQ_Contact(in1 := #iState, in2 := #READ_REGS_NEXT)
      wire#w3
      { S7_Templates := "SrcType := DInt" } GE_Contact(in1 := #iCurrentRegisterReadIndex, in2 := #iNumReadRegisters)
      Move(in := #WRITE_REGS_INIT, out1 => #iNextState)
   END_RUNG
   RUNG wire#w3
      { S7_Templates := "SrcType := DInt" } LT_Contact(in1 := #iCurrentRegisterReadIndex, in2 := #iNumReadRegisters)
      { S7_Templates := "DestType := DInt" } Inc( #iCurrentRegisterReadIndex )
      Move(in := #READ_REGS, out1 => #iNextState)
   END_RUNG
   RUNG wire#powerrail
      { S7_Templates := "SrcType := Int" } EQ_Contact(in1 := #iState, in2 := #WRITE_REGS_NEXT)
      wire#w4
      { S7_Templates := "SrcType := DInt" } GE_Contact(in1 := #iCurrentRegisterWriteIndex, in2 := #iNumWriteRegisters)
      Move(in := #IDLE, out1 => #iNextState)
   END_RUNG
   RUNG wire#w4
      { S7_Templates := "SrcType := DInt" } LT_Contact(in1 := #iCurrentRegisterWriteIndex, in2 := #iNumWriteRegisters)
      { S7_Templates := "DestType := DInt" } Inc( #iCurrentRegisterWriteIndex )
      Move(in := #WRITE_REGS, out1 => #iNextState)
   END_RUNG
   // the same network as SCL:
   #_w1 := #iState = #READ_DISC_NEXT;
   IF #_w1 AND (#iCurrentDiscreteReadIndex >= #iNumReadDiscrete) THEN
       #iNextState := #WRITE_COILS_INIT;
   END_IF;
   #_w2 := #_w1 AND (#iCurrentDiscreteReadIndex < #iNumReadDiscrete);
   IF #_w2 THEN
       #iCurrentDiscreteReadIndex := #iCurrentDiscreteReadIndex + 1;
       #iNextState := #READ_DISC;
   END_IF;
   #_w3 := #iState = #WRITE_COILS_NEXT;
   IF #_w3 AND (#iCurrentCoilWriteIndex >= #iNumWriteCoils) THEN #iNextState := #READ_REGS_INIT; END_IF;
   #_w4 := #_w3 AND (#iCurrentCoilWriteIndex < #iNumWriteCoils);
   IF #_w4 THEN
       #iCurrentCoilWriteIndex := #iCurrentCoilWriteIndex + 1;
       #iNextState := #WRITE_COILS;
   END_IF;
   #_w5 := #iState = #READ_REGS_NEXT;
   IF #_w5 AND (#iCurrentRegisterReadIndex >= #iNumReadRegisters) THEN
       #iNextState := #WRITE_REGS_INIT;
   END_IF;
   #_w6 := #_w5 AND (#iCurrentRegisterReadIndex < #iNumReadRegisters);
   IF #_w6 THEN
       #iCurrentRegisterReadIndex := #iCurrentRegisterReadIndex + 1;
       #iNextState := #READ_REGS;
   END_IF;
   #_w7 := #iState = #WRITE_REGS_NEXT;
   IF #_w7 AND (#iCurrentRegisterWriteIndex >= #iNumWriteRegisters) THEN #iNextState := #IDLE; END_IF;
   #_w8 := #_w7 AND (#iCurrentRegisterWriteIndex < #iNumWriteRegisters);
   IF #_w8 THEN
       #iCurrentRegisterWriteIndex := #iCurrentRegisterWriteIndex + 1;
       #iNextState := #WRITE_REGS;
   END_IF;
END_REGION

REGION Network 7: ------------------------------ Configure settings and call MB_CLIENT ----------------------------------
END_REGION

REGION Network 8: Set register and data bytes based on array index
   // Assuming that all input address data is formatted with full Modbus address offsets, i.e. coils (00001), discrete inputs (10001), input registers (30001), holding registers (40001)
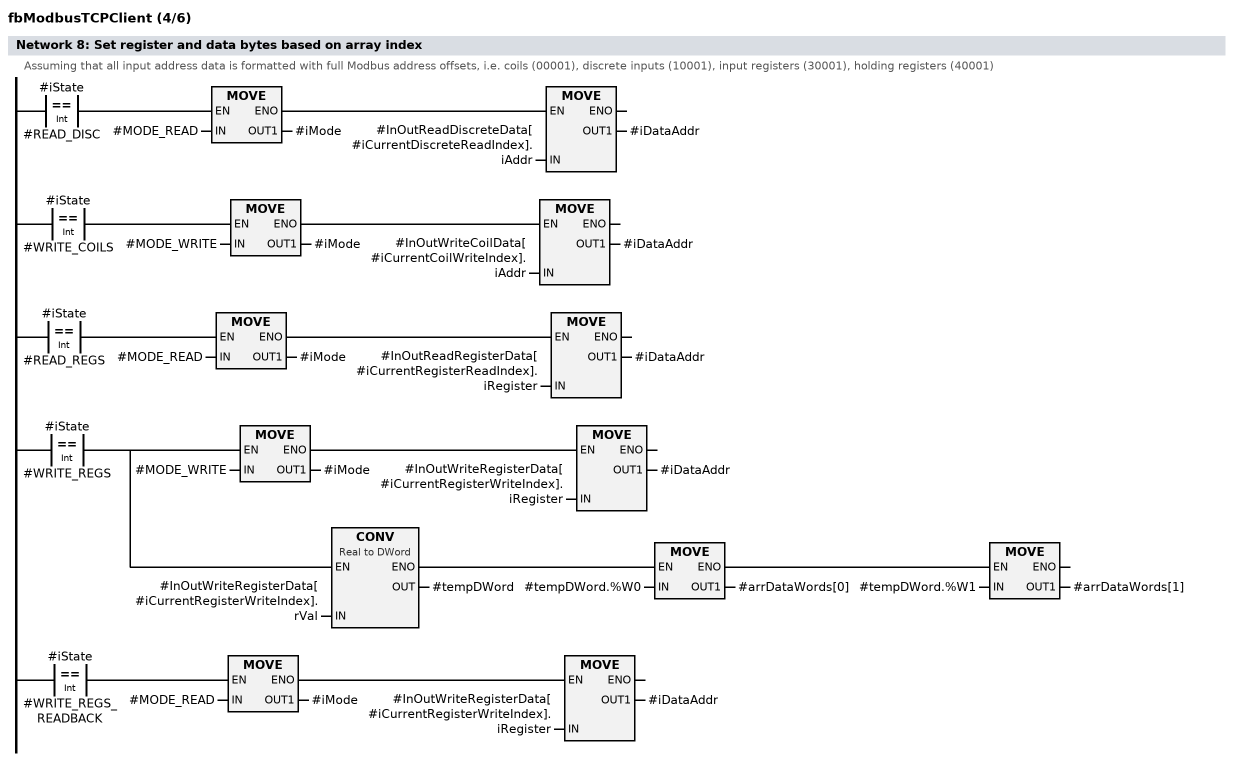
   RUNG wire#powerrail
      { S7_Templates := "SrcType := Int" } EQ_Contact(in1 := #iState, in2 := #READ_DISC)
      Move(in := #MODE_READ, out1 => #iMode)
      Move(in := #InOutReadDiscreteData[#iCurrentDiscreteReadIndex].iAddr, out1 => #iDataAddr)
   END_RUNG
   RUNG wire#powerrail
      { S7_Templates := "SrcType := Int" } EQ_Contact(in1 := #iState, in2 := #WRITE_COILS)
      Move(in := #MODE_WRITE, out1 => #iMode)
      Move(in := #InOutWriteCoilData[#iCurrentCoilWriteIndex].iAddr, out1 => #iDataAddr)
   END_RUNG
   RUNG wire#powerrail
      { S7_Templates := "SrcType := Int" } EQ_Contact(in1 := #iState, in2 := #READ_REGS)
      Move(in := #MODE_READ, out1 => #iMode)
      Move(in := #InOutReadRegisterData[#iCurrentRegisterReadIndex].iRegister, out1 => #iDataAddr)
   END_RUNG
   RUNG wire#powerrail
      { S7_Templates := "SrcType := Int" } EQ_Contact(in1 := #iState, in2 := #WRITE_REGS)
      wire#w1
      Move(in := #MODE_WRITE, out1 => #iMode)
      Move(in := #InOutWriteRegisterData[#iCurrentRegisterWriteIndex].iRegister, out1 => #iDataAddr)
   END_RUNG
   RUNG wire#w1
      { S7_Templates := "[SrcType := Real, DestType := DWord]" } Convert(in := #InOutWriteRegisterData[#iCurrentRegisterWriteIndex].rVal, out => #tempDWord)
      Move(in := #tempDWord.%W0, out1 => #arrDataWords[0])
      Move(in := #tempDWord.%W1, out1 => #arrDataWords[1])
   END_RUNG
   RUNG wire#powerrail
      { S7_Templates := "SrcType := Int" } EQ_Contact(in1 := #iState, in2 := #WRITE_REGS_READBACK)
      Move(in := #MODE_READ, out1 => #iMode)
      Move(in := #InOutWriteRegisterData[#iCurrentRegisterWriteIndex].iRegister, out1 => #iDataAddr)
   END_RUNG
   // the same network as SCL:
   IF #iState = #READ_DISC THEN
       #iMode := #MODE_READ;
       #iDataAddr := #InOutReadDiscreteData[#iCurrentDiscreteReadIndex].iAddr;
   END_IF;
   IF #iState = #WRITE_COILS THEN
       #iMode := #MODE_WRITE;
       #iDataAddr := #InOutWriteCoilData[#iCurrentCoilWriteIndex].iAddr;
   END_IF;
   IF #iState = #READ_REGS THEN
       #iMode := #MODE_READ;
       #iDataAddr := #InOutReadRegisterData[#iCurrentRegisterReadIndex].iRegister;
   END_IF;
   IF #iState = #WRITE_REGS THEN
       #iMode := #MODE_WRITE;
       #iDataAddr := #InOutWriteRegisterData[#iCurrentRegisterWriteIndex].iRegister;
       #tempDWord := REAL_TO_DWORD(#InOutWriteRegisterData[#iCurrentRegisterWriteIndex].rVal);
       #arrDataWords[0] := #tempDWord.%W0;
       #arrDataWords[1] := #tempDWord.%W1;
   END_IF;
   IF #iState = #WRITE_REGS_READBACK THEN
       #iMode := #MODE_READ;
       #iDataAddr := #InOutWriteRegisterData[#iCurrentRegisterWriteIndex].iRegister;
   END_IF;
END_REGION

REGION Network 9: MB_CLIENT block call
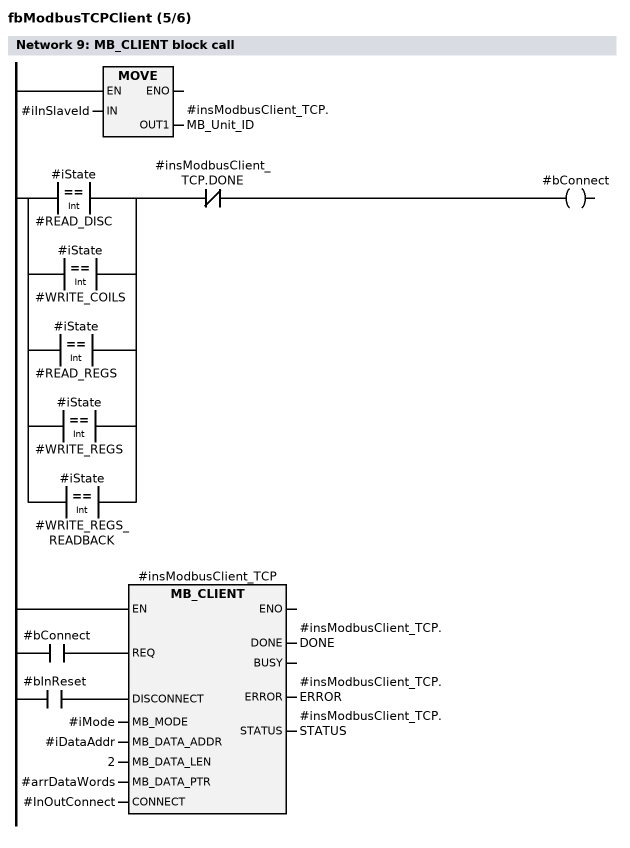
   RUNG wire#powerrail
      Move(in := #iInSlaveId, out1 => #insModbusClient_TCP.MB_Unit_ID)
   END_RUNG
   RUNG wire#powerrail
      { S7_Templates := "SrcType := Int" } EQ_Contact(in1 := #iState, in2 := #READ_DISC)
      wire#w1
      I_Contact( #insModbusClient_TCP.DONE )
      Coil( #bConnect )
   END_RUNG
   RUNG wire#powerrail
      { S7_Templates := "SrcType := Int" } EQ_Contact(in1 := #iState, in2 := #WRITE_COILS)
   END_RUNG wire#w1
   RUNG wire#powerrail
      { S7_Templates := "SrcType := Int" } EQ_Contact(in1 := #iState, in2 := #READ_REGS)
   END_RUNG wire#w1
   RUNG wire#powerrail
      { S7_Templates := "SrcType := Int" } EQ_Contact(in1 := #iState, in2 := #WRITE_REGS)
   END_RUNG wire#w1
   RUNG wire#powerrail
      { S7_Templates := "SrcType := Int" } EQ_Contact(in1 := #iState, in2 := #WRITE_REGS_READBACK)
   END_RUNG wire#w1
   RUNG wire#powerrail
      #insModbusClient_TCP.MB_CLIENT(REQ := wire#w2, DISCONNECT := wire#w3, MB_MODE := #iMode, MB_DATA_ADDR := #iDataAddr, MB_DATA_LEN := 2, MB_DATA_PTR := #arrDataWords, CONNECT := #InOutConnect, DONE => #insModbusClient_TCP.DONE, BUSY =>, ERROR => #insModbusClient_TCP.ERROR, STATUS => #insModbusClient_TCP.STATUS)
   END_RUNG
   RUNG wire#powerrail
      Contact( #bConnect )
   END_RUNG wire#w2
   RUNG wire#powerrail
      Contact( #bInReset )
   END_RUNG wire#w3
   // the same network as SCL:
   #insModbusClient_TCP.MB_Unit_ID := #iInSlaveId;
   #bConnect := ((#iState = #READ_DISC) OR (#iState = #WRITE_COILS) OR (#iState = #READ_REGS) OR (#iState = #WRITE_REGS) OR (#iState = #WRITE_REGS_READBACK)) AND NOT #insModbusClient_TCP.DONE;
   #insModbusClient_TCP(REQ := #bConnect,   // MB_CLIENT
                        DISCONNECT := #bInReset,
                        MB_MODE := #iMode,
                        MB_DATA_ADDR := #iDataAddr,
                        MB_DATA_LEN := 2,
                        MB_DATA_PTR := #arrDataWords,
                        CONNECT := #InOutConnect,
                        DONE => #insModbusClient_TCP.DONE,
                        ERROR => #insModbusClient_TCP.ERROR,
                        STATUS => #insModbusClient_TCP.STATUS);
END_REGION

REGION Network 10: Set error status
   // Ignore error code 16#80A3 (same connection already being used)
   // Go back to idle if stuck waiting for read/write
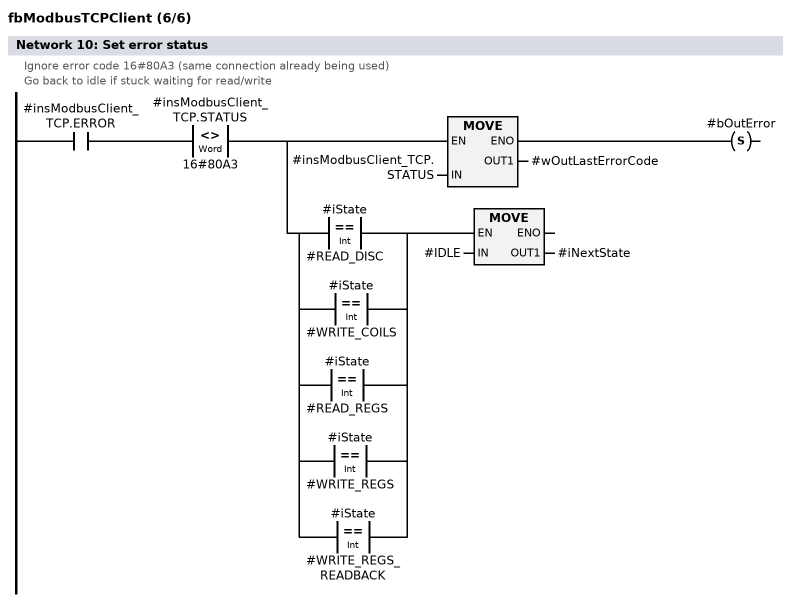
   RUNG wire#powerrail
      Contact( #insModbusClient_TCP.ERROR )
      { S7_Templates := "SrcType := Word" } NE_Contact(in1 := #insModbusClient_TCP.STATUS, in2 := 16#80A3)
      wire#w1
      Move(in := #insModbusClient_TCP.STATUS, out1 => #wOutLastErrorCode)
      S_Coil( #bOutError )
   END_RUNG
   RUNG wire#w1
      { S7_Templates := "SrcType := Int" } EQ_Contact(in1 := #iState, in2 := #READ_DISC)
      wire#w2
      Move(in := #IDLE, out1 => #iNextState)
   END_RUNG
   RUNG wire#w1
      { S7_Templates := "SrcType := Int" } EQ_Contact(in1 := #iState, in2 := #WRITE_COILS)
   END_RUNG wire#w2
   RUNG wire#w1
      { S7_Templates := "SrcType := Int" } EQ_Contact(in1 := #iState, in2 := #READ_REGS)
   END_RUNG wire#w2
   RUNG wire#w1
      { S7_Templates := "SrcType := Int" } EQ_Contact(in1 := #iState, in2 := #WRITE_REGS)
   END_RUNG wire#w2
   RUNG wire#w1
      { S7_Templates := "SrcType := Int" } EQ_Contact(in1 := #iState, in2 := #WRITE_REGS_READBACK)
   END_RUNG wire#w2
   // the same network as SCL:
   #_w1 := #insModbusClient_TCP.ERROR AND (#insModbusClient_TCP.STATUS <> 16#80A3);
   IF #_w1 THEN
       #wOutLastErrorCode := #insModbusClient_TCP.STATUS;
       #bOutError := TRUE;
   END_IF;
   IF #_w1 AND ((#iState = #READ_DISC) OR (#iState = #WRITE_COILS) OR (#iState = #READ_REGS) OR (#iState = #WRITE_REGS) OR (#iState = #WRITE_REGS_READBACK)) THEN
       #iNextState := #IDLE;
   END_IF;
END_REGION
END_FUNCTION_BLOCK

FUNCTION_BLOCK "fbRoomCO2Control"   // FB13, LAD
{ S7_Optimized_Access := 'TRUE' }
VERSION : 0.1
// stored: AutoNumber true, IsIECCheckEnabled false, IsRetainMemResEnabled false, MemoryReserve 100, SetENOAutomatically false, UDAEnableTagReadback false
   VAR_INPUT
      iInCO2ReadingRaw { ExternalAccessible := 'False'; ExternalVisible := 'False'; ExternalWritable := 'False'} : Int;
   END_VAR
   VAR_OUTPUT
      bOutSolenoid { ExternalAccessible := 'False'; ExternalVisible := 'False'; ExternalWritable := 'False'} : Bool;
   END_VAR
   VAR
      AI_CO2Sensor { ExternalVisible := 'False'} : "fbAlarmedSetpoint";
   END_VAR
   VAR RETAIN
      Controls { ExternalVisible := 'False'} : Struct
         iModeCommand { ExternalVisible := 'False'} : Int;   // 0: Off, 1: Periodic Dosing
         tMeasurementInterval { ExternalVisible := 'False'} : Time := T#30s;   // Time between measurements
         tDosingDuration { ExternalVisible := 'False'} : Time := T#5s;   // Time to open solenoid if measurement is below setpoint
      END_STRUCT;
   END_VAR
   VAR
      Status { ExternalVisible := 'False'; ExternalWritable := 'False'} : Struct
         tElapsedMeasurement { ExternalVisible := 'False'; ExternalWritable := 'False'} : Time;
         tElapsedDosing { ExternalVisible := 'False'; ExternalWritable := 'False'} : Time;
      END_STRUCT;
   END_VAR
   VAR RETAIN
      TON_MeasurementCycle { ExternalAccessible := 'False'; ExternalVisible := 'False'; ExternalWritable := 'False'} : TON_TIME;
      TP_Dosing { ExternalAccessible := 'False'; ExternalVisible := 'False'; ExternalWritable := 'False'} : TP_TIME;
   END_VAR
   VAR_TEMP
      bCheckMeasurement : Bool;
   END_VAR
   VAR CONSTANT
      eMode_Off : Int := 0;   // forced off
      eMode_PeriodicDosing : Int := 2;   // auto
   END_VAR
   // AI_CO2Sensor.arrSetpoints[1].rSetpoint := 400.0;
   // AI_CO2Sensor.Config.rHighCalibration := 10000.0;
BEGIN

REGION Network 1 (SCL)
   // process CO2 sensor input
   #AI_CO2Sensor(#iInCO2ReadingRaw);

   // if mode is set to periodic dosing, run timer to periodically check value
   #bCheckMeasurement := #TON_MeasurementCycle.Q;
   #TON_MeasurementCycle(IN := #Controls.iModeCommand = #eMode_PeriodicDosing AND NOT #bCheckMeasurement,
                         PT := #Controls.tMeasurementInterval,
                         ET => #Status.tElapsedMeasurement);

   //if value is below setpoint, open valve for set duration
   #TP_Dosing(IN := #bCheckMeasurement AND #AI_CO2Sensor.rActual < #AI_CO2Sensor.rSetpoint,
               PT := #Controls.tDosingDuration,
               Q => #bOutSolenoid,
               ET => #Status.tElapsedDosing);
END_REGION
END_FUNCTION_BLOCK

FUNCTION "fcAnalogInput" : Real
{ S7_Optimized_Access := 'TRUE' }
VERSION : 0.1
   VAR_INPUT 
      iInRawValue : Int;
      rLowCalibration : Real;
      rHighCalibration : Real;
   END_VAR


BEGIN
	// Scale raw input (0 to 27648 for 4-20mA and 0-10V)
	#fcAnalogInput :=
	
	( INT_TO_REAL(#iInRawValue) / INT_TO_REAL("IoScaling.S7Analog.Default.iRawMax")) *
	(#rHighCalibration - #rLowCalibration) + #rLowCalibration;
	
END_FUNCTION
